LIN {X 0,Y 413.384,Z 401.555,A -85,B 0,C 180,E1 -10493.04,E2 -10493.04} C_VEL
LIN {X 0,Y 413.39,Z 404.987,A -85,B 0,C 180,E1 -10494.691,E2 -10494.691} C_VEL
LIN {X 0,Y 412.815,Z 411.314,A -85,B 0,C 180,E1 -10497.573,E2 -10497.573} C_VEL
LIN {X 0,Y 412.207,Z 419.076,A -85,B 0,C 180,E1 -10500.936,E2 -10500.936} C_VEL
LIN {X 0,Y 411.681,Z 426.853,A -85,B 0,C 180,E1 -10504.197,E2 -10504.197} C_VEL
LIN {X 0,Y 411.179,Z 436.082,A -85,B 0,C 180,E1 -10507.914,E2 -10507.914} C_VEL
LIN {X 0,Y 410.861,Z 444.017,A -85,B 0,C 180,E1 -10511.036,E2 -10511.036} C_VEL
LIN {X 0,Y 410.682,Z 447.705,A -85,B 0,C 180,E1 -10512.405,E2 -10512.405} C_VEL
LIN {X 0,Y 412.802,Z 461.15,A -85,B 0,C 180,E1 -10512.893,E2 -10512.893} C_VEL
LIN {X 0,Y 414.62,Z 474.244,A -85,B 0,C 180,E1 -10513.572,E2 -10513.572} C_VEL
LIN {X 0,Y 414.778,Z 478.671,A -85,B 0,C 180,E1 -10513.831,E2 -10513.831} C_VEL
LIN {X 0,Y 413.979,Z 490.398,A -85,B 0,C 180,E1 -10514.62,E2 -10514.62} C_VEL
LIN {X 0,Y 413.231,Z 501.649,A -85,B 0,C 180,E1 -10515.59,E2 -10515.59} C_VEL
LIN {X 0,Y 412.528,Z 512,A -85,B 0,C 180,E1 -10516.706,E2 -10516.706} C_VEL
LIN {X 0,Y 411.827,Z 521.233,A -85,B 0,C 180,E1 -10517.935,E2 -10517.935} C_VEL
LIN {X 0,Y 411.123,Z 530.239,A -85,B 0,C 180,E1 -10519.413,E2 -10519.413} C_VEL
LIN {X 0,Y 410.679,Z 537.503,A -85,B 0,C 180,E1 -10520.894,E2 -10520.894} C_VEL
LIN {X 0,Y 410.352,Z 542.408,A -85,B 0,C 180,E1 -10522.127,E2 -10522.127} C_VEL
LIN {X 0,Y 410.175,Z 547.189,A -85,B 0,C 180,E1 -10523.608,E2 -10523.608} C_VEL
LIN {X 0,Y 410.096,Z 550.845,A -85,B 0,C 180,E1 -10525.086,E2 -10525.086} C_VEL
LIN {X 0,Y 409.955,Z 552.727,A -85,B 0,C 180,E1 -10526.07,E2 -10526.07} C_VEL
LIN {X 0,Y 410.007,Z 554.15,A -85,B 0,C 180,E1 -10527.054,E2 -10527.054} C_VEL
LIN {X 0,Y 409.988,Z 555.163,A -85,B 0,C 180,E1 -10528.037,E2 -10528.037} C_VEL
LIN {X 0,Y 409.959,Z 555.783,A -85,B 0,C 180,E1 -10529.02,E2 -10529.02} C_VEL
LIN {X 0,Y 409.967,Z 556.008,A -85,B 0,C 180,E1 -10530.002,E2 -10530.002} C_VEL
LIN {X 0,Y 409.959,Z 555.794,A -85,B 0,C 180,E1 -10530.984,E2 -10530.984} C_VEL
LIN {X 0,Y 409.989,Z 555.187,A -85,B 0,C 180,E1 -10531.967,E2 -10531.967} C_VEL
LIN {X 0,Y 410.008,Z 554.186,A -85,B 0,C 180,E1 -10532.949,E2 -10532.949} C_VEL
LIN {X 0,Y 409.955,Z 552.774,A -85,B 0,C 180,E1 -10533.934,E2 -10533.934} C_VEL
LIN {X 0,Y 410.109,Z 549.821,A -85,B 0,C 180,E1 -10535.41,E2 -10535.41} C_VEL
LIN {X 0,Y 410.2,Z 545.812,A -85,B 0,C 180,E1 -10536.89,E2 -10536.89} C_VEL
LIN {X 0,Y 410.553,Z 539.656,A -85,B 0,C 180,E1 -10538.616,E2 -10538.616} C_VEL
LIN {X 0,Y 410.995,Z 532.935,A -85,B 0,C 180,E1 -10540.096,E2 -10540.096} C_VEL
LIN {X 0,Y 411.586,Z 524.602,A -85,B 0,C 180,E1 -10541.576,E2 -10541.576} C_VEL
LIN {X 0,Y 412.261,Z 516.065,A -85,B 0,C 180,E1 -10542.806,E2 -10542.806} C_VEL
LIN {X 0,Y 412.962,Z 505.339,A -85,B 0,C 180,E1 -10544.056,E2 -10544.056} C_VEL
LIN {X 0,Y 413.802,Z 493.67,A -85,B 0,C 180,E1 -10545.139,E2 -10545.139} C_VEL
LIN {X 0,Y 414.646,Z 481.768,A -85,B 0,C 180,E1 -10545.988,E2 -10545.988} C_VEL
LIN {X 0,Y 414.818,Z 475.494,A -85,B 0,C 180,E1 -10546.359,E2 -10546.359} C_VEL
LIN {X 0,Y 413.068,Z 462.585,A -85,B 0,C 180,E1 -10547.042,E2 -10547.042} C_VEL
LIN {X 0,Y 410.836,Z 449.124,A -85,B 0,C 180,E1 -10547.554,E2 -10547.554} C_VEL
LIN {X 0,Y 410.721,Z 447.803,A -85,B 0,C 180,E1 -10547.635,E2 -10547.635} C_VEL
LIN {X 0,Y 411.094,Z 439.097,A -85,B 0,C 180,E1 -10551.041,E2 -10551.041} C_VEL
LIN {X 0,Y 411.483,Z 431.213,A -85,B 0,C 180,E1 -10554.201,E2 -10554.201} C_VEL
LIN {X 0,Y 411.896,Z 424.656,A -85,B 0,C 180,E1 -10556.884,E2 -10556.884} C_VEL
LIN {X 0,Y 412.427,Z 416.854,A -85,B 0,C 180,E1 -10560.18,E2 -10560.18} C_VEL
LIN {X 0,Y 413.084,Z 409.18,A -85,B 0,C 180,E1 -10563.523,E2 -10563.523} C_VEL
LIN {X 0,Y 413.51,Z 403.963,A -85,B 0,C 180,E1 -10565.9,E2 -10565.9} C_VEL
LIN {X 0,Y 413.155,Z 400.089,A -85,B 0,C 180,E1 -10567.763,E2 -10567.763} C_VEL
LIN {X 0,Y 411.926,Z 393.158,A -85,B 0,C 180,E1 -10571.349,E2 -10571.349} C_VEL
LIN {X 0,Y 411.183,Z 389.269,A -85,B 0,C 180,E1 -10573.596,E2 -10573.596} C_VEL
LIN {X 0,Y 411.179,Z 389.27,A -85,B 0,C 180,E1 -10576.867,E2 -10576.867} C_VEL
LIN {X 0,Y 411.215,Z 389.263,A -85,B 0,C 180,E1 -10580.273,E2 -10580.273} C_VEL
LIN {X 0,Y 411.198,Z 389.264,A -85,B 0,C 180,E1 -10583.448,E2 -10583.448} C_VEL
LIN {X 0,Y 411.213,Z 389.265,A -85,B 0,C 180,E1 -10586.874,E2 -10586.874} C_VEL
LIN {X 0,Y 411.239,Z 389.262,A -85,B 0,C 180,E1 -10590.645,E2 -10590.645} C_VEL
LIN {X 0,Y 411.244,Z 389.257,A -85,B 0,C 180,E1 -10593.619,E2 -10593.619} C_VEL
LIN {X 0,Y 411.209,Z 389.265,A -85,B 0,C 180,E1 -10596.853,E2 -10596.853} C_VEL
LIN {X 0,Y 411.221,Z 389.263,A -85,B 0,C 180,E1 -10600.051,E2 -10600.051} C_VEL
LIN {X 0,Y 411.269,Z 389.255,A -85,B 0,C 180,E1 -10603.131,E2 -10603.131} C_VEL
LIN {X 0,Y 411.311,Z 389.25,A -85,B 0,C 180,E1 -10606.896,E2 -10606.896} C_VEL
LIN {X 0,Y 411.298,Z 389.255,A -85,B 0,C 180,E1 -10610.161,E2 -10610.161} C_VEL
LIN {X 0,Y 411.458,Z 389.23,A -85,B 0,C 180,E1 -10613.133,E2 -10613.133} C_VEL
LIN {X 0,Y 411.313,Z 389.249,A -85,B 0,C 180,E1 -10615.099,E2 -10615.099} C_VEL
LIN {X 0,Y 411.516,Z 389.228,A -85,B 0,C 180,E1 -10618.042,E2 -10618.042} C_VEL
LIN {X 0,Y 411.645,Z 389.212,A -85,B 0,C 180,E1 -10620,E2 -10620} C_VEL
LIN {X 0,Y 411.462,Z 389.23,A -85,B 0,C 180,E1 -10622.937,E2 -10622.937} C_VEL
LIN {X 0,Y 411.464,Z 389.23,A -85,B 0,C 180,E1 -10626.867,E2 -10626.867} C_VEL
LIN {X 0,Y 411.36,Z 389.242,A -85,B 0,C 180,E1 -10628.845,E2 -10628.845} C_VEL
LIN {X 0,Y 411.289,Z 389.256,A -85,B 0,C 180,E1 -10631.833,E2 -10631.833} C_VEL
LIN {X 0,Y 411.265,Z 389.255,A -85,B 0,C 180,E1 -10634.852,E2 -10634.852} C_VEL
LIN {X 0,Y 411.258,Z 389.259,A -85,B 0,C 180,E1 -10637.915,E2 -10637.915} C_VEL
LIN {X 0,Y 411.202,Z 389.264,A -85,B 0,C 180,E1 -10641.034,E2 -10641.034} C_VEL
LIN {X 0,Y 411.232,Z 389.26,A -85,B 0,C 180,E1 -10644.215,E2 -10644.215} C_VEL
LIN {X 0,Y 411.265,Z 389.259,A -85,B 0,C 180,E1 -10647.477,E2 -10647.477} C_VEL
LIN {X 0,Y 411.195,Z 389.264,A -85,B 0,C 180,E1 -10650.847,E2 -10650.847} C_VEL
LIN {X 0,Y 411.211,Z 389.262,A -85,B 0,C 180,E1 -10654.333,E2 -10654.333} C_VEL
LIN {X 0,Y 411.2,Z 389.264,A -85,B 0,C 180,E1 -10657.973,E2 -10657.973} C_VEL
LIN {X 0,Y 411.187,Z 389.265,A -85,B 0,C 180,E1 -10660.504,E2 -10660.504} C_VEL
LIN {X 0,Y 411.179,Z 389.269,A -85,B 0,C 180,E1 -10663.133,E2 -10663.133} C_VEL
LIN {X 0,Y 411.173,Z 389.266,A -85,B 0,C 180,E1 -10665.88,E2 -10665.88} C_VEL
LIN {X 0,Y 411.169,Z 389.269,A -85,B 0,C 180,E1 -10668.771,E2 -10668.771} C_VEL
LIN {X 0,Y 411.211,Z 389.262,A -85,B 0,C 180,E1 -10671.83,E2 -10671.83} C_VEL
LIN {X 0,Y 411.216,Z 389.265,A -85,B 0,C 180,E1 -10675.121,E2 -10675.121} C_VEL
LIN {X 0,Y 411.171,Z 389.266,A -85,B 0,C 180,E1 -10678.002,E2 -10678.002} C_VEL
LIN {X 0,Y 411.223,Z 389.261,A -85,B 0,C 180,E1 -10681.409,E2 -10681.409} C_VEL
LIN {X 0,Y 411.243,Z 389.257,A -85,B 0,C 180,E1 -10683.618,E2 -10683.618} C_VEL
LIN {X 0,Y 411.208,Z 389.266,A -85,B 0,C 180,E1 -10686.851,E2 -10686.851} C_VEL
LIN {X 0,Y 411.22,Z 389.261,A -85,B 0,C 180,E1 -10690.049,E2 -10690.049} C_VEL
LIN {X 0,Y 411.268,Z 389.257,A -85,B 0,C 180,E1 -10693.13,E2 -10693.13} C_VEL
LIN {X 0,Y 411.236,Z 389.261,A -85,B 0,C 180,E1 -10696.156,E2 -10696.156} C_VEL
LIN {X 0,Y 411.194,Z 389.266,A -85,B 0,C 180,E1 -10698.163,E2 -10698.163} C_VEL
LIN {X 0,Y 410.866,Z 389.309,A -85,B 0,C 180,E1 -10701.142,E2 -10701.142} C_VEL
LIN {X 0,Y 410.774,Z 389.525,A -85,B 0,C 180,E1 -10702.131,E2 -10702.131} C_VEL
LIN {X 0,Y 410.784,Z 392.396,A -85,B 0,C 180,E1 -10705.091,E2 -10705.091} C_VEL
LIN {X 0,Y 410.551,Z 394.344,A -85,B 0,C 180,E1 -10707.054,E2 -10707.054} C_VEL
LIN {X 0,Y 410.411,Z 397.302,A -85,B 0,C 180,E1 -10709.998,E2 -10709.998} C_VEL
LIN {X 0,Y 410.505,Z 401.242,A -85,B 0,C 180,E1 -10713.925,E2 -10713.925} C_VEL
LIN {X 0,Y 410.425,Z 402.961,A -85,B 0,C 180,E1 -10715.556,E2 -10715.556} C_VEL
LIN {X 0,Y 414.064,Z 417.484,A -85,B 0,C 180,E1 -10716.24,E2 -10716.24} C_VEL
LIN {X 0,Y 415.548,Z 425.03,A -85,B 0,C 180,E1 -10716.675,E2 -10716.675} C_VEL
LIN {X 0,Y 414.873,Z 437.253,A -85,B 0,C 180,E1 -10717.42,E2 -10717.42} C_VEL
LIN {X 0,Y 414.236,Z 448.24,A -85,B 0,C 180,E1 -10718.29,E2 -10718.29} C_VEL
LIN {X 0,Y 413.445,Z 458.989,A -85,B 0,C 180,E1 -10719.36,E2 -10719.36} C_VEL
LIN {X 0,Y 412.757,Z 468.534,A -85,B 0,C 180,E1 -10720.545,E2 -10720.545} C_VEL
LIN {X 0,Y 412.152,Z 476.118,A -85,B 0,C 180,E1 -10721.683,E2 -10721.683} C_VEL
LIN {X 0,Y 411.15,Z 479.89,A -85,B 0,C 180,E1 -10722.305,E2 -10722.305} C_VEL
LIN {X 0,Y 407.883,Z 485.677,A -85,B 0,C 180,E1 -10723.336,E2 -10723.336} C_VEL
LIN {X 0,Y 404.703,Z 490.822,A -85,B 0,C 180,E1 -10724.443,E2 -10724.443} C_VEL
LIN {X 0,Y 403.848,Z 493.53,A -85,B 0,C 180,E1 -10725.177,E2 -10725.177} C_VEL
LIN {X 0,Y 403.486,Z 498.112,A -85,B 0,C 180,E1 -10726.664,E2 -10726.664} C_VEL
LIN {X 0,Y 403.2,Z 501.878,A -85,B 0,C 180,E1 -10728.283,E2 -10728.283} C_VEL
LIN {X 0,Y 403.025,Z 504.16,A -85,B 0,C 180,E1 -10729.668,E2 -10729.668} C_VEL
LIN {X 0,Y 402.881,Z 506,A -85,B 0,C 180,E1 -10731.487,E2 -10731.487} C_VEL
LIN {X 0,Y 402.85,Z 506.437,A -85,B 0,C 180,E1 -10732.567,E2 -10732.567} C_VEL
LIN {X 0,Y 402.857,Z 506.444,A -85,B 0,C 180,E1 -10733.653,E2 -10733.653} C_VEL
LIN {X 0,Y 402.893,Z 505.879,A -85,B 0,C 180,E1 -10734.895,E2 -10734.895} C_VEL
LIN {X 0,Y 402.978,Z 505.025,A -85,B 0,C 180,E1 -10735.846,E2 -10735.846} C_VEL
LIN {X 0,Y 403.169,Z 503.115,A -85,B 0,C 180,E1 -10737.249,E2 -10737.249} C_VEL
LIN {X 0,Y 403.388,Z 500.443,A -85,B 0,C 180,E1 -10738.625,E2 -10738.625} C_VEL
LIN {X 0,Y 403.718,Z 495.928,A -85,B 0,C 180,E1 -10740.318,E2 -10740.318} C_VEL
LIN {X 0,Y 404.191,Z 490.125,A -85,B 0,C 180,E1 -10741.966,E2 -10741.966} C_VEL
LIN {X 0,Y 404.843,Z 482.961,A -85,B 0,C 180,E1 -10743.564,E2 -10743.564} C_VEL
LIN {X 0,Y 405.459,Z 475.593,A -85,B 0,C 180,E1 -10744.887,E2 -10744.887} C_VEL
LIN {X 0,Y 406.229,Z 466.736,A -85,B 0,C 180,E1 -10746.181,E2 -10746.181} C_VEL
LIN {X 0,Y 407.033,Z 456.303,A -85,B 0,C 180,E1 -10747.415,E2 -10747.415} C_VEL
LIN {X 0,Y 407.848,Z 444.851,A -85,B 0,C 180,E1 -10748.492,E2 -10748.492} C_VEL
LIN {X 0,Y 408.543,Z 433.308,A -85,B 0,C 180,E1 -10749.333,E2 -10749.333} C_VEL
LIN {X 0,Y 408.71,Z 425.291,A -85,B 0,C 180,E1 -10749.813,E2 -10749.813} C_VEL
LIN {X 0,Y 405.684,Z 412.827,A -85,B 0,C 180,E1 -10750.529,E2 -10750.529} C_VEL
LIN {X 0,Y 403.305,Z 404.188,A -85,B 0,C 180,E1 -10750.941,E2 -10750.941} C_VEL
LIN {X 0,Y 403.412,Z 400.785,A -85,B 0,C 180,E1 -10754.416,E2 -10754.416} C_VEL
LIN {X 0,Y 403.442,Z 398.12,A -85,B 0,C 180,E1 -10757.204,E2 -10757.204} C_VEL
LIN {X 0,Y 403.54,Z 395.443,A -85,B 0,C 180,E1 -10760.018,E2 -10760.018} C_VEL
LIN {X 0,Y 403.676,Z 391.997,A -85,B 0,C 180,E1 -10763.705,E2 -10763.705} C_VEL
LIN {X 0,Y 403.734,Z 390.847,A -85,B 0,C 180,E1 -10764.939,E2 -10764.939} C_VEL
LIN {X 0,Y 403.891,Z 390.181,A -85,B 0,C 180,E1 -10766.635,E2 -10766.635} C_VEL
LIN {X 0,Y 404.121,Z 390.15,A -85,B 0,C 180,E1 -10769.713,E2 -10769.713} C_VEL
LIN {X 0,Y 404.178,Z 390.14,A -85,B 0,C 180,E1 -10773.122,E2 -10773.122} C_VEL
LIN {X 0,Y 404.167,Z 390.144,A -85,B 0,C 180,E1 -10776.425,E2 -10776.425} C_VEL
LIN {X 0,Y 404.208,Z 390.134,A -85,B 0,C 180,E1 -10779.859,E2 -10779.859} C_VEL
LIN {X 0,Y 404.196,Z 390.139,A -85,B 0,C 180,E1 -10782.992,E2 -10782.992} C_VEL
LIN {X 0,Y 404.262,Z 390.128,A -85,B 0,C 180,E1 -10786.938,E2 -10786.938} C_VEL
LIN {X 0,Y 404.252,Z 390.129,A -85,B 0,C 180,E1 -10789.988,E2 -10789.988} C_VEL
LIN {X 0,Y 404.393,Z 390.11,A -85,B 0,C 180,E1 -10793.013,E2 -10793.013} C_VEL
LIN {X 0,Y 404.272,Z 390.129,A -85,B 0,C 180,E1 -10795.014,E2 -10795.014} C_VEL
LIN {X 0,Y 404.464,Z 390.106,A -85,B 0,C 180,E1 -10798.009,E2 -10798.009} C_VEL
LIN {X 0,Y 404.592,Z 390.088,A -85,B 0,C 180,E1 -10800,E2 -10800} C_VEL
LIN {X 0,Y 404.411,Z 390.11,A -85,B 0,C 180,E1 -10802.989,E2 -10802.989} C_VEL
LIN {X 0,Y 404.391,Z 390.113,A -85,B 0,C 180,E1 -10806.988,E2 -10806.988} C_VEL
LIN {X 0,Y 404.251,Z 390.132,A -85,B 0,C 180,E1 -10810.012,E2 -10810.012} C_VEL
LIN {X 0,Y 404.247,Z 390.132,A -85,B 0,C 180,E1 -10813.212,E2 -10813.212} C_VEL
LIN {X 0,Y 404.196,Z 390.139,A -85,B 0,C 180,E1 -10817.008,E2 -10817.008} C_VEL
LIN {X 0,Y 404.189,Z 390.139,A -85,B 0,C 180,E1 -10820.35,E2 -10820.35} C_VEL
LIN {X 0,Y 404.167,Z 390.144,A -85,B 0,C 180,E1 -10823.575,E2 -10823.575} C_VEL
LIN {X 0,Y 404.179,Z 390.143,A -85,B 0,C 180,E1 -10826.878,E2 -10826.878} C_VEL
LIN {X 0,Y 404.129,Z 390.149,A -85,B 0,C 180,E1 -10830.287,E2 -10830.287} C_VEL
LIN {X 0,Y 404.129,Z 390.147,A -85,B 0,C 180,E1 -10833.814,E2 -10833.814} C_VEL
LIN {X 0,Y 404.126,Z 390.147,A -85,B 0,C 180,E1 -10836.878,E2 -10836.878} C_VEL
LIN {X 0,Y 404.154,Z 390.147,A -85,B 0,C 180,E1 -10840.085,E2 -10840.085} C_VEL
LIN {X 0,Y 404.192,Z 390.146,A -85,B 0,C 180,E1 -10843.094,E2 -10843.094} C_VEL
LIN {X 0,Y 404.219,Z 390.214,A -85,B 0,C 180,E1 -10845.98,E2 -10845.98} C_VEL
LIN {X 0,Y 405.367,Z 396.616,A -85,B 0,C 180,E1 -10849.716,E2 -10849.716} C_VEL
LIN {X 0,Y 406.32,Z 402.279,A -85,B 0,C 180,E1 -10852.747,E2 -10852.747} C_VEL
LIN {X 0,Y 406.437,Z 405.532,A -85,B 0,C 180,E1 -10854.362,E2 -10854.362} C_VEL
LIN {X 0,Y 405.804,Z 412.364,A -85,B 0,C 180,E1 -10857.531,E2 -10857.531} C_VEL
LIN {X 0,Y 405.153,Z 420.058,A -85,B 0,C 180,E1 -10860.944,E2 -10860.944} C_VEL
LIN {X 0,Y 404.633,Z 427.83,A -85,B 0,C 180,E1 -10864.267,E2 -10864.267} C_VEL
LIN {X 0,Y 404.089,Z 437.021,A -85,B 0,C 180,E1 -10868.044,E2 -10868.044} C_VEL
LIN {X 0,Y 403.742,Z 444.938,A -85,B 0,C 180,E1 -10871.217,E2 -10871.217} C_VEL
LIN {X 0,Y 403.641,Z 447.176,A -85,B 0,C 180,E1 -10872.08,E2 -10872.08} C_VEL
LIN {X 0,Y 405.791,Z 460.799,A -85,B 0,C 180,E1 -10872.589,E2 -10872.589} C_VEL
LIN {X 0,Y 407.58,Z 473.449,A -85,B 0,C 180,E1 -10873.259,E2 -10873.259} C_VEL
LIN {X 0,Y 407.981,Z 477.702,A -85,B 0,C 180,E1 -10873.519,E2 -10873.519} C_VEL
LIN {X 0,Y 407.115,Z 489.968,A -85,B 0,C 180,E1 -10874.354,E2 -10874.354} C_VEL
LIN {X 0,Y 406.286,Z 501.704,A -85,B 0,C 180,E1 -10875.386,E2 -10875.386} C_VEL
LIN {X 0,Y 405.587,Z 511.564,A -85,B 0,C 180,E1 -10876.474,E2 -10876.474} C_VEL
LIN {X 0,Y 404.868,Z 520.796,A -85,B 0,C 180,E1 -10877.725,E2 -10877.725} C_VEL
LIN {X 0,Y 404.1,Z 529.801,A -85,B 0,C 180,E1 -10879.227,E2 -10879.227} C_VEL
LIN {X 0,Y 403.61,Z 537.065,A -85,B 0,C 180,E1 -10880.733,E2 -10880.733} C_VEL
LIN {X 0,Y 403.299,Z 541.973,A -85,B 0,C 180,E1 -10881.988,E2 -10881.988} C_VEL
LIN {X 0,Y 403.069,Z 547.202,A -85,B 0,C 180,E1 -10883.652,E2 -10883.652} C_VEL
LIN {X 0,Y 403.008,Z 550.411,A -85,B 0,C 180,E1 -10885,E2 -10885} C_VEL
LIN {X 0,Y 402.877,Z 552.295,A -85,B 0,C 180,E1 -10886.001,E2 -10886.001} C_VEL
LIN {X 0,Y 402.909,Z 553.717,A -85,B 0,C 180,E1 -10887.002,E2 -10887.002} C_VEL
LIN {X 0,Y 402.921,Z 554.733,A -85,B 0,C 180,E1 -10888.003,E2 -10888.003} C_VEL
LIN {X 0,Y 402.884,Z 555.353,A -85,B 0,C 180,E1 -10889.002,E2 -10889.002} C_VEL
LIN {X 0,Y 402.89,Z 555.578,A -85,B 0,C 180,E1 -10890.002,E2 -10890.002} C_VEL
LIN {X 0,Y 402.921,Z 554.757,A -85,B 0,C 180,E1 -10892.001,E2 -10892.001} C_VEL
LIN {X 0,Y 402.91,Z 553.754,A -85,B 0,C 180,E1 -10893.001,E2 -10893.001} C_VEL
LIN {X 0,Y 402.878,Z 552.343,A -85,B 0,C 180,E1 -10894.003,E2 -10894.003} C_VEL
LIN {X 0,Y 403.007,Z 549.387,A -85,B 0,C 180,E1 -10895.506,E2 -10895.506} C_VEL
LIN {X 0,Y 403.118,Z 545.377,A -85,B 0,C 180,E1 -10897.012,E2 -10897.012} C_VEL
LIN {X 0,Y 403.518,Z 539.219,A -85,B 0,C 180,E1 -10898.768,E2 -10898.768} C_VEL
LIN {X 0,Y 403.967,Z 532.495,A -85,B 0,C 180,E1 -10900.274,E2 -10900.274} C_VEL
LIN {X 0,Y 404.6,Z 524.161,A -85,B 0,C 180,E1 -10901.779,E2 -10901.779} C_VEL
LIN {X 0,Y 405.266,Z 515.617,A -85,B 0,C 180,E1 -10903.031,E2 -10903.031} C_VEL
LIN {X 0,Y 405.984,Z 505.786,A -85,B 0,C 180,E1 -10904.205,E2 -10904.205} C_VEL
LIN {X 0,Y 406.807,Z 494.65,A -85,B 0,C 180,E1 -10905.277,E2 -10905.277} C_VEL
LIN {X 0,Y 407.657,Z 483.352,A -85,B 0,C 180,E1 -10906.134,E2 -10906.134} C_VEL
LIN {X 0,Y 407.882,Z 475.699,A -85,B 0,C 180,E1 -10906.607,E2 -10906.607} C_VEL
LIN {X 0,Y 406.106,Z 462.732,A -85,B 0,C 180,E1 -10907.316,E2 -10907.316} C_VEL
LIN {X 0,Y 403.985,Z 449.659,A -85,B 0,C 180,E1 -10907.838,E2 -10907.838} C_VEL
LIN {X 0,Y 403.644,Z 447.403,A -85,B 0,C 180,E1 -10907.938,E2 -10907.938} C_VEL
LIN {X 0,Y 404.013,Z 440.038,A -85,B 0,C 180,E1 -10910.894,E2 -10910.894} C_VEL
LIN {X 0,Y 404.394,Z 432.159,A -85,B 0,C 180,E1 -10914.106,E2 -10914.106} C_VEL
LIN {X 0,Y 404.897,Z 424.569,A -85,B 0,C 180,E1 -10917.284,E2 -10917.284} C_VEL
LIN {X 0,Y 405.5,Z 416.561,A -85,B 0,C 180,E1 -10920.751,E2 -10920.751} C_VEL
LIN {X 0,Y 406.127,Z 409.667,A -85,B 0,C 180,E1 -10923.835,E2 -10923.835} C_VEL
LIN {X 0,Y 406.507,Z 404.99,A -85,B 0,C 180,E1 -10926.004,E2 -10926.004} C_VEL
LIN {X 0,Y 406.143,Z 401.148,A -85,B 0,C 180,E1 -10927.902,E2 -10927.902} C_VEL
LIN {X 0,Y 405.017,Z 394.766,A -85,B 0,C 180,E1 -10931.255,E2 -10931.255} C_VEL
LIN {X 0,Y 404.143,Z 390.145,A -85,B 0,C 180,E1 -10933.875,E2 -10933.875} C_VEL
LIN {X 0,Y 404.142,Z 390.146,A -85,B 0,C 180,E1 -10937.296,E2 -10937.296} C_VEL
LIN {X 0,Y 404.176,Z 390.14,A -85,B 0,C 180,E1 -10939.956,E2 -10939.956} C_VEL
LIN {X 0,Y 404.142,Z 390.145,A -85,B 0,C 180,E1 -10943.126,E2 -10943.126} C_VEL
LIN {X 0,Y 404.15,Z 390.142,A -85,B 0,C 180,E1 -10946.188,E2 -10946.188} C_VEL
LIN {X 0,Y 404.152,Z 390.14,A -85,B 0,C 180,E1 -10949.715,E2 -10949.715} C_VEL
LIN {X 0,Y 404.202,Z 390.136,A -85,B 0,C 180,E1 -10953.123,E2 -10953.123} C_VEL
LIN {X 0,Y 404.183,Z 390.137,A -85,B 0,C 180,E1 -10955.335,E2 -10955.335} C_VEL
LIN {X 0,Y 404.145,Z 390.146,A -85,B 0,C 180,E1 -10958.581,E2 -10958.581} C_VEL
LIN {X 0,Y 404.216,Z 390.133,A -85,B 0,C 180,E1 -10961.762,E2 -10961.762} C_VEL
LIN {X 0,Y 404.212,Z 390.135,A -85,B 0,C 180,E1 -10964.882,E2 -10964.882} C_VEL
LIN {X 0,Y 404.262,Z 390.13,A -85,B 0,C 180,E1 -10967.959,E2 -10967.959} C_VEL
LIN {X 0,Y 404.411,Z 390.113,A -85,B 0,C 180,E1 -10972.129,E2 -10972.129} C_VEL
LIN {X 0,Y 404.425,Z 390.111,A -85,B 0,C 180,E1 -10974.015,E2 -10974.015} C_VEL
LIN {X 0,Y 404.485,Z 390.103,A -85,B 0,C 180,E1 -10978.008,E2 -10978.008} C_VEL
LIN {X 0,Y 404.614,Z 390.087,A -85,B 0,C 180,E1 -10980,E2 -10980} C_VEL
LIN {X 0,Y 404.42,Z 390.107,A -85,B 0,C 180,E1 -10982.988,E2 -10982.988} C_VEL
LIN {X 0,Y 404.415,Z 390.107,A -85,B 0,C 180,E1 -10986.987,E2 -10986.987} C_VEL
LIN {X 0,Y 404.264,Z 390.131,A -85,B 0,C 180,E1 -10990.012,E2 -10990.012} C_VEL
LIN {X 0,Y 404.272,Z 390.126,A -85,B 0,C 180,E1 -10993.211,E2 -10993.211} C_VEL
LIN {X 0,Y 404.222,Z 390.132,A -85,B 0,C 180,E1 -10997.007,E2 -10997.007} C_VEL
LIN {X 0,Y 404.169,Z 390.139,A -85,B 0,C 180,E1 -11000.351,E2 -11000.351} C_VEL
LIN {X 0,Y 404.175,Z 390.142,A -85,B 0,C 180,E1 -11003.574,E2 -11003.574} C_VEL
LIN {X 0,Y 404.19,Z 390.14,A -85,B 0,C 180,E1 -11005.766,E2 -11005.766} C_VEL
LIN {X 0,Y 404.201,Z 390.136,A -85,B 0,C 180,E1 -11007.999,E2 -11007.999} C_VEL
LIN {X 0,Y 404.145,Z 390.146,A -85,B 0,C 180,E1 -11011.557,E2 -11011.557} C_VEL
LIN {X 0,Y 404.19,Z 390.139,A -85,B 0,C 180,E1 -11015.016,E2 -11015.016} C_VEL
LIN {X 0,Y 404.16,Z 390.141,A -85,B 0,C 180,E1 -11018.756,E2 -11018.756} C_VEL
LIN {X 0,Y 404.129,Z 390.146,A -85,B 0,C 180,E1 -11021.599,E2 -11021.599} C_VEL
LIN {X 0,Y 404.151,Z 390.141,A -85,B 0,C 180,E1 -11024.521,E2 -11024.521} C_VEL
LIN {X 0,Y 404.142,Z 390.146,A -85,B 0,C 180,E1 -11027.295,E2 -11027.295} C_VEL
LIN {X 0,Y 404.175,Z 390.138,A -85,B 0,C 180,E1 -11029.955,E2 -11029.955} C_VEL
LIN {X 0,Y 404.142,Z 390.146,A -85,B 0,C 180,E1 -11033.124,E2 -11033.124} C_VEL
LIN {X 0,Y 404.15,Z 390.141,A -85,B 0,C 180,E1 -11036.187,E2 -11036.187} C_VEL
LIN {X 0,Y 404.151,Z 390.141,A -85,B 0,C 180,E1 -11039.714,E2 -11039.714} C_VEL
LIN {X 0,Y 404.201,Z 390.138,A -85,B 0,C 180,E1 -11043.122,E2 -11043.122} C_VEL
LIN {X 0,Y 404.182,Z 390.138,A -85,B 0,C 180,E1 -11045.333,E2 -11045.333} C_VEL
LIN {X 0,Y 404.144,Z 390.146,A -85,B 0,C 180,E1 -11048.579,E2 -11048.579} C_VEL
LIN {X 0,Y 404.215,Z 390.133,A -85,B 0,C 180,E1 -11051.761,E2 -11051.761} C_VEL
LIN {X 0,Y 404.21,Z 390.137,A -85,B 0,C 180,E1 -11054.881,E2 -11054.881} C_VEL
LIN {X 0,Y 404.165,Z 390.14,A -85,B 0,C 180,E1 -11057.954,E2 -11057.954} C_VEL
LIN {X 0,Y 403.858,Z 390.182,A -85,B 0,C 180,E1 -11060.988,E2 -11060.988} C_VEL
LIN {X 0,Y 403.721,Z 390.231,A -85,B 0,C 180,E1 -11061.993,E2 -11061.993} C_VEL
LIN {X 0,Y 403.735,Z 393.111,A -85,B 0,C 180,E1 -11065.005,E2 -11065.005} C_VEL
LIN {X 0,Y 403.509,Z 395.091,A -85,B 0,C 180,E1 -11067.003,E2 -11067.003} C_VEL
LIN {X 0,Y 403.352,Z 398.094,A -85,B 0,C 180,E1 -11069.998,E2 -11069.998} C_VEL
LIN {X 0,Y 403.435,Z 401.056,A -85,B 0,C 180,E1 -11072.994,E2 -11072.994} C_VEL
LIN {X 0,Y 403.359,Z 403.34,A -85,B 0,C 180,E1 -11075.246,E2 -11075.246} C_VEL
LIN {X 0,Y 406.893,Z 417.253,A -85,B 0,C 180,E1 -11075.915,E2 -11075.915} C_VEL
LIN {X 0,Y 408.648,Z 425.75,A -85,B 0,C 180,E1 -11076.416,E2 -11076.416} C_VEL
LIN {X 0,Y 408.042,Z 437.83,A -85,B 0,C 180,E1 -11077.171,E2 -11077.171} C_VEL
LIN {X 0,Y 407.365,Z 448.794,A -85,B 0,C 180,E1 -11078.056,E2 -11078.056} C_VEL
LIN {X 0,Y 406.593,Z 459.049,A -85,B 0,C 180,E1 -11079.09,E2 -11079.09} C_VEL
LIN {X 0,Y 405.901,Z 468.13,A -85,B 0,C 180,E1 -11080.221,E2 -11080.221} C_VEL
LIN {X 0,Y 405.178,Z 476.751,A -85,B 0,C 180,E1 -11081.529,E2 -11081.529} C_VEL
LIN {X 0,Y 404.509,Z 484.878,A -85,B 0,C 180,E1 -11083.051,E2 -11083.051} C_VEL
LIN {X 0,Y 403.993,Z 491.499,A -85,B 0,C 180,E1 -11084.608,E2 -11084.608} C_VEL
LIN {X 0,Y 403.848,Z 493.53,A -85,B 0,C 180,E1 -11085.177,E2 -11085.177} C_VEL
LIN {X 0,Y 402.993,Z 496.078,A -85,B 0,C 180,E1 -11085.931,E2 -11085.931} C_VEL
LIN {X 0,Y 399.834,Z 499.728,A -85,B 0,C 180,E1 -11087.169,E2 -11087.169} C_VEL
LIN {X 0,Y 396.728,Z 502.721,A -85,B 0,C 180,E1 -11088.458,E2 -11088.458} C_VEL
LIN {X 0,Y 395.963,Z 504.065,A -85,B 0,C 180,E1 -11089.281,E2 -11089.281} C_VEL
LIN {X 0,Y 395.82,Z 505.911,A -85,B 0,C 180,E1 -11090.798,E2 -11090.798} C_VEL
LIN {X 0,Y 395.787,Z 506.87,A -85,B 0,C 180,E1 -11092.577,E2 -11092.577} C_VEL
LIN {X 0,Y 395.776,Z 506.754,A -85,B 0,C 180,E1 -11094.103,E2 -11094.103} C_VEL
LIN {X 0,Y 395.855,Z 506.098,A -85,B 0,C 180,E1 -11095.217,E2 -11095.217} C_VEL
LIN {X 0,Y 395.956,Z 504.986,A -85,B 0,C 180,E1 -11096.34,E2 -11096.34} C_VEL
LIN {X 0,Y 396.239,Z 502.315,A -85,B 0,C 180,E1 -11098.032,E2 -11098.032} C_VEL
LIN {X 0,Y 396.53,Z 498.365,A -85,B 0,C 180,E1 -11099.75,E2 -11099.75} C_VEL
LIN {X 0,Y 396.96,Z 493.376,A -85,B 0,C 180,E1 -11101.37,E2 -11101.37} C_VEL
LIN {X 0,Y 397.552,Z 487.256,A -85,B 0,C 180,E1 -11102.926,E2 -11102.926} C_VEL
LIN {X 0,Y 398.151,Z 480.117,A -85,B 0,C 180,E1 -11104.389,E2 -11104.389} C_VEL
LIN {X 0,Y 398.993,Z 471.02,A -85,B 0,C 180,E1 -11105.879,E2 -11105.879} C_VEL
LIN {X 0,Y 399.821,Z 461.214,A -85,B 0,C 180,E1 -11107.171,E2 -11107.171} C_VEL
LIN {X 0,Y 400.62,Z 451.62,A -85,B 0,C 180,E1 -11108.195,E2 -11108.195} C_VEL
LIN {X 0,Y 401.439,Z 440.118,A -85,B 0,C 180,E1 -11109.178,E2 -11109.178} C_VEL
LIN {X 0,Y 402.044,Z 427.299,A -85,B 0,C 180,E1 -11110.016,E2 -11110.016} C_VEL
LIN {X 0,Y 399.094,Z 414.764,A -85,B 0,C 180,E1 -11110.78,E2 -11110.78} C_VEL
LIN {X 0,Y 396.262,Z 404.634,A -85,B 0,C 180,E1 -11111.281,E2 -11111.281} C_VEL
LIN {X 0,Y 396.361,Z 401.217,A -85,B 0,C 180,E1 -11114.826,E2 -11114.826} C_VEL
LIN {X 0,Y 396.417,Z 398.088,A -85,B 0,C 180,E1 -11118.121,E2 -11118.121} C_VEL
LIN {X 0,Y 396.52,Z 394.824,A -85,B 0,C 180,E1 -11121.659,E2 -11121.659} C_VEL
LIN {X 0,Y 396.667,Z 392.103,A -85,B 0,C 180,E1 -11124.583,E2 -11124.583} C_VEL
LIN {X 0,Y 396.68,Z 391.311,A -85,B 0,C 180,E1 -11125.463,E2 -11125.463} C_VEL
LIN {X 0,Y 397.013,Z 391.038,A -85,B 0,C 180,E1 -11128.174,E2 -11128.174} C_VEL
LIN {X 0,Y 397.098,Z 391.022,A -85,B 0,C 180,E1 -11131.455,E2 -11131.455} C_VEL
LIN {X 0,Y 397.135,Z 391.018,A -85,B 0,C 180,E1 -11134.486,E2 -11134.486} C_VEL
LIN {X 0,Y 397.158,Z 391.015,A -85,B 0,C 180,E1 -11138.185,E2 -11138.185} C_VEL
LIN {X 0,Y 397.152,Z 391.015,A -85,B 0,C 180,E1 -11141.426,E2 -11141.426} C_VEL
LIN {X 0,Y 397.16,Z 391.014,A -85,B 0,C 180,E1 -11144.607,E2 -11144.607} C_VEL
LIN {X 0,Y 397.21,Z 391.007,A -85,B 0,C 180,E1 -11147.742,E2 -11147.742} C_VEL
LIN {X 0,Y 397.375,Z 390.986,A -85,B 0,C 180,E1 -11152.04,E2 -11152.04} C_VEL
LIN {X 0,Y 397.244,Z 391.004,A -85,B 0,C 180,E1 -11154.925,E2 -11154.925} C_VEL
LIN {X 0,Y 397.432,Z 390.982,A -85,B 0,C 180,E1 -11157.973,E2 -11157.973} C_VEL
LIN {X 0,Y 397.562,Z 390.963,A -85,B 0,C 180,E1 -11160,E2 -11160} C_VEL
LIN {X 0,Y 397.369,Z 390.988,A -85,B 0,C 180,E1 -11163.042,E2 -11163.042} C_VEL
LIN {X 0,Y 397.344,Z 390.991,A -85,B 0,C 180,E1 -11167.112,E2 -11167.112} C_VEL
LIN {X 0,Y 397.209,Z 391.01,A -85,B 0,C 180,E1 -11170.191,E2 -11170.191} C_VEL
LIN {X 0,Y 397.207,Z 391.008,A -85,B 0,C 180,E1 -11173.322,E2 -11173.322} C_VEL
LIN {X 0,Y 397.163,Z 391.015,A -85,B 0,C 180,E1 -11177.156,E2 -11177.156} C_VEL
LIN {X 0,Y 397.14,Z 391.018,A -85,B 0,C 180,E1 -11180.728,E2 -11180.728} C_VEL
LIN {X 0,Y 397.124,Z 391.022,A -85,B 0,C 180,E1 -11184.019,E2 -11184.019} C_VEL
LIN {X 0,Y 397.177,Z 391.015,A -85,B 0,C 180,E1 -11187.392,E2 -11187.392} C_VEL
LIN {X 0,Y 397.062,Z 391.029,A -85,B 0,C 180,E1 -11190.884,E2 -11190.884} C_VEL
LIN {X 0,Y 397.11,Z 391.022,A -85,B 0,C 180,E1 -11194.495,E2 -11194.495} C_VEL
LIN {X 0,Y 397.095,Z 391.024,A -85,B 0,C 180,E1 -11198.276,E2 -11198.276} C_VEL
LIN {X 0,Y 397.144,Z 391.022,A -85,B 0,C 180,E1 -11201.995,E2 -11201.995} C_VEL
LIN {X 0,Y 397.17,Z 391.082,A -85,B 0,C 180,E1 -11205.569,E2 -11205.569} C_VEL
LIN {X 0,Y 398.022,Z 396.038,A -85,B 0,C 180,E1 -11208.573,E2 -11208.573} C_VEL
LIN {X 0,Y 399.129,Z 402.093,A -85,B 0,C 180,E1 -11211.958,E2 -11211.958} C_VEL
LIN {X 0,Y 399.47,Z 406.118,A -85,B 0,C 180,E1 -11214.027,E2 -11214.027} C_VEL
LIN {X 0,Y 398.915,Z 412.102,A -85,B 0,C 180,E1 -11216.9,E2 -11216.9} C_VEL
LIN {X 0,Y 398.189,Z 419.758,A -85,B 0,C 180,E1 -11220.386,E2 -11220.386} C_VEL
LIN {X 0,Y 397.657,Z 427.498,A -85,B 0,C 180,E1 -11223.782,E2 -11223.782} C_VEL
LIN {X 0,Y 397.122,Z 435.319,A -85,B 0,C 180,E1 -11227.089,E2 -11227.089} C_VEL
LIN {X 0,Y 396.721,Z 444.514,A -85,B 0,C 180,E1 -11230.871,E2 -11230.871} C_VEL
LIN {X 0,Y 396.597,Z 446.645,A -85,B 0,C 180,E1 -11231.736,E2 -11231.736} C_VEL
LIN {X 0,Y 398.896,Z 460.907,A -85,B 0,C 180,E1 -11232.294,E2 -11232.294} C_VEL
LIN {X 0,Y 400.636,Z 473.751,A -85,B 0,C 180,E1 -11232.998,E2 -11232.998} C_VEL
LIN {X 0,Y 401.026,Z 479.493,A -85,B 0,C 180,E1 -11233.367,E2 -11233.367} C_VEL
LIN {X 0,Y 400.139,Z 491.152,A -85,B 0,C 180,E1 -11234.205,E2 -11234.205} C_VEL
LIN {X 0,Y 399.255,Z 502.632,A -85,B 0,C 180,E1 -11235.267,E2 -11235.267} C_VEL
LIN {X 0,Y 398.455,Z 513.253,A -85,B 0,C 180,E1 -11236.508,E2 -11236.508} C_VEL
LIN {X 0,Y 397.739,Z 522.003,A -85,B 0,C 180,E1 -11237.76,E2 -11237.76} C_VEL
LIN {X 0,Y 396.978,Z 530.698,A -85,B 0,C 180,E1 -11239.289,E2 -11239.289} C_VEL
LIN {X 0,Y 396.496,Z 537.664,A -85,B 0,C 180,E1 -11240.823,E2 -11240.823} C_VEL
LIN {X 0,Y 396.138,Z 543.253,A -85,B 0,C 180,E1 -11242.356,E2 -11242.356} C_VEL
LIN {X 0,Y 395.949,Z 547.646,A -85,B 0,C 180,E1 -11243.889,E2 -11243.889} C_VEL
LIN {X 0,Y 395.921,Z 549.978,A -85,B 0,C 180,E1 -11244.91,E2 -11244.91} C_VEL
LIN {X 0,Y 395.802,Z 551.863,A -85,B 0,C 180,E1 -11245.929,E2 -11245.929} C_VEL
LIN {X 0,Y 395.812,Z 553.284,A -85,B 0,C 180,E1 -11246.949,E2 -11246.949} C_VEL
LIN {X 0,Y 395.854,Z 554.303,A -85,B 0,C 180,E1 -11247.967,E2 -11247.967} C_VEL
LIN {X 0,Y 395.813,Z 554.924,A -85,B 0,C 180,E1 -11248.985,E2 -11248.985} C_VEL
LIN {X 0,Y 395.815,Z 555.148,A -85,B 0,C 180,E1 -11250.002,E2 -11250.002} C_VEL
LIN {X 0,Y 395.855,Z 554.327,A -85,B 0,C 180,E1 -11252.037,E2 -11252.037} C_VEL
LIN {X 0,Y 395.813,Z 553.323,A -85,B 0,C 180,E1 -11253.055,E2 -11253.055} C_VEL
LIN {X 0,Y 395.803,Z 551.912,A -85,B 0,C 180,E1 -11254.075,E2 -11254.075} C_VEL
LIN {X 0,Y 395.908,Z 548.952,A -85,B 0,C 180,E1 -11255.605,E2 -11255.605} C_VEL
LIN {X 0,Y 396.063,Z 544.943,A -85,B 0,C 180,E1 -11257.137,E2 -11257.137} C_VEL
LIN {X 0,Y 396.46,Z 538.781,A -85,B 0,C 180,E1 -11258.925,E2 -11258.925} C_VEL
LIN {X 0,Y 396.915,Z 532.054,A -85,B 0,C 180,E1 -11260.458,E2 -11260.458} C_VEL
LIN {X 0,Y 397.595,Z 523.719,A -85,B 0,C 180,E1 -11261.989,E2 -11261.989} C_VEL
LIN {X 0,Y 398.301,Z 515.171,A -85,B 0,C 180,E1 -11263.263,E2 -11263.263} C_VEL
LIN {X 0,Y 399.097,Z 504.859,A -85,B 0,C 180,E1 -11264.508,E2 -11264.508} C_VEL
LIN {X 0,Y 399.944,Z 494.199,A -85,B 0,C 180,E1 -11265.546,E2 -11265.546} C_VEL
LIN {X 0,Y 400.824,Z 482.989,A -85,B 0,C 180,E1 -11266.41,E2 -11266.41} C_VEL
LIN {X 0,Y 401.098,Z 477.767,A -85,B 0,C 180,E1 -11266.746,E2 -11266.746} C_VEL
LIN {X 0,Y 399.452,Z 464.949,A -85,B 0,C 180,E1 -11267.496,E2 -11267.496} C_VEL
LIN {X 0,Y 397.268,Z 451.221,A -85,B 0,C 180,E1 -11268.089,E2 -11268.089} C_VEL
LIN {X 0,Y 396.609,Z 447.084,A -85,B 0,C 180,E1 -11268.234,E2 -11268.234} C_VEL
LIN {X 0,Y 397.042,Z 438.345,A -85,B 0,C 180,E1 -11271.823,E2 -11271.823} C_VEL
LIN {X 0,Y 397.628,Z 429.242,A -85,B 0,C 180,E1 -11275.655,E2 -11275.655} C_VEL
LIN {X 0,Y 398.174,Z 421.406,A -85,B 0,C 180,E1 -11279.04,E2 -11279.04} C_VEL
LIN {X 0,Y 398.774,Z 414.326,A -85,B 0,C 180,E1 -11282.226,E2 -11282.226} C_VEL
LIN {X 0,Y 399.456,Z 407.289,A -85,B 0,C 180,E1 -11285.494,E2 -11285.494} C_VEL
LIN {X 0,Y 399.466,Z 404.726,A -85,B 0,C 180,E1 -11286.741,E2 -11286.741} C_VEL
LIN {X 0,Y 398.668,Z 399.608,A -85,B 0,C 180,E1 -11289.394,E2 -11289.394} C_VEL
LIN {X 0,Y 397.56,Z 393.337,A -85,B 0,C 180,E1 -11292.851,E2 -11292.851} C_VEL
LIN {X 0,Y 397.106,Z 391.023,A -85,B 0,C 180,E1 -11294.271,E2 -11294.271} C_VEL
LIN {X 0,Y 397.075,Z 391.027,A -85,B 0,C 180,E1 -11297.733,E2 -11297.733} C_VEL
LIN {X 0,Y 397.133,Z 391.018,A -85,B 0,C 180,E1 -11301.14,E2 -11301.14} C_VEL
LIN {X 0,Y 397.125,Z 391.019,A -85,B 0,C 180,E1 -11304.497,E2 -11304.497} C_VEL
LIN {X 0,Y 397.084,Z 391.021,A -85,B 0,C 180,E1 -11307.929,E2 -11307.929} C_VEL
LIN {X 0,Y 397.128,Z 391.015,A -85,B 0,C 180,E1 -11311.457,E2 -11311.457} C_VEL
LIN {X 0,Y 397.159,Z 391.016,A -85,B 0,C 180,E1 -11314.488,E2 -11314.488} C_VEL
LIN {X 0,Y 397.115,Z 391.018,A -85,B 0,C 180,E1 -11317.086,E2 -11317.086} C_VEL
LIN {X 0,Y 397.154,Z 391.016,A -85,B 0,C 180,E1 -11320.353,E2 -11320.353} C_VEL
LIN {X 0,Y 397.173,Z 391.01,A -85,B 0,C 180,E1 -11323.553,E2 -11323.553} C_VEL
LIN {X 0,Y 397.235,Z 391.005,A -85,B 0,C 180,E1 -11326.703,E2 -11326.703} C_VEL
LIN {X 0,Y 397.223,Z 391.005,A -85,B 0,C 180,E1 -11329.809,E2 -11329.809} C_VEL
LIN {X 0,Y 397.355,Z 390.987,A -85,B 0,C 180,E1 -11332.888,E2 -11332.888} C_VEL
LIN {X 0,Y 397.257,Z 391,A -85,B 0,C 180,E1 -11334.925,E2 -11334.925} C_VEL
LIN {X 0,Y 397.454,Z 390.979,A -85,B 0,C 180,E1 -11337.973,E2 -11337.973} C_VEL
LIN {X 0,Y 397.584,Z 390.963,A -85,B 0,C 180,E1 -11340,E2 -11340} C_VEL
LIN {X 0,Y 397.379,Z 390.984,A -85,B 0,C 180,E1 -11343.041,E2 -11343.041} C_VEL
LIN {X 0,Y 397.368,Z 390.985,A -85,B 0,C 180,E1 -11347.112,E2 -11347.112} C_VEL
LIN {X 0,Y 397.223,Z 391.007,A -85,B 0,C 180,E1 -11350.191,E2 -11350.191} C_VEL
LIN {X 0,Y 397.233,Z 391.004,A -85,B 0,C 180,E1 -11353.321,E2 -11353.321} C_VEL
LIN {X 0,Y 397.188,Z 391.009,A -85,B 0,C 180,E1 -11357.155,E2 -11357.155} C_VEL
LIN {X 0,Y 397.108,Z 391.018,A -85,B 0,C 180,E1 -11360.73,E2 -11360.73} C_VEL
LIN {X 0,Y 397.139,Z 391.016,A -85,B 0,C 180,E1 -11364.018,E2 -11364.018} C_VEL
LIN {X 0,Y 397.2,Z 391.011,A -85,B 0,C 180,E1 -11367.39,E2 -11367.39} C_VEL
LIN {X 0,Y 397.084,Z 391.022,A -85,B 0,C 180,E1 -11370.882,E2 -11370.882} C_VEL
LIN {X 0,Y 397.131,Z 391.015,A -85,B 0,C 180,E1 -11374.493,E2 -11374.493} C_VEL
LIN {X 0,Y 397.108,Z 391.018,A -85,B 0,C 180,E1 -11378.274,E2 -11378.274} C_VEL
LIN {X 0,Y 397.094,Z 391.022,A -85,B 0,C 180,E1 -11380.908,E2 -11380.908} C_VEL
LIN {X 0,Y 397.107,Z 391.02,A -85,B 0,C 180,E1 -11383.648,E2 -11383.648} C_VEL
LIN {X 0,Y 397.107,Z 391.018,A -85,B 0,C 180,E1 -11386.52,E2 -11386.52} C_VEL
LIN {X 0,Y 397.12,Z 391.017,A -85,B 0,C 180,E1 -11390.422,E2 -11390.422} C_VEL
LIN {X 0,Y 397.114,Z 391.018,A -85,B 0,C 180,E1 -11394.264,E2 -11394.264} C_VEL
LIN {X 0,Y 397.12,Z 391.02,A -85,B 0,C 180,E1 -11396.726,E2 -11396.726} C_VEL
LIN {X 0,Y 397.13,Z 391.016,A -85,B 0,C 180,E1 -11400.295,E2 -11400.295} C_VEL
LIN {X 0,Y 397.2,Z 391.01,A -85,B 0,C 180,E1 -11402.609,E2 -11402.609} C_VEL
LIN {X 0,Y 397.138,Z 391.014,A -85,B 0,C 180,E1 -11405.98,E2 -11405.98} C_VEL
LIN {X 0,Y 397.144,Z 391.013,A -85,B 0,C 180,E1 -11409.703,E2 -11409.703} C_VEL
LIN {X 0,Y 397.186,Z 391.012,A -85,B 0,C 180,E1 -11412.843,E2 -11412.843} C_VEL
LIN {X 0,Y 397.171,Z 391.01,A -85,B 0,C 180,E1 -11415.655,E2 -11415.655} C_VEL
LIN {X 0,Y 397.127,Z 391.016,A -85,B 0,C 180,E1 -11417.737,E2 -11417.737} C_VEL
LIN {X 0,Y 396.827,Z 391.058,A -85,B 0,C 180,E1 -11420.826,E2 -11420.826} C_VEL
LIN {X 0,Y 396.697,Z 391.076,A -85,B 0,C 180,E1 -11421.85,E2 -11421.85} C_VEL
LIN {X 0,Y 396.688,Z 393.859,A -85,B 0,C 180,E1 -11424.916,E2 -11424.916} C_VEL
LIN {X 0,Y 396.469,Z 395.834,A -85,B 0,C 180,E1 -11426.95,E2 -11426.95} C_VEL
LIN {X 0,Y 396.287,Z 398.835,A -85,B 0,C 180,E1 -11429.998,E2 -11429.998} C_VEL
LIN {X 0,Y 396.39,Z 401.899,A -85,B 0,C 180,E1 -11433.047,E2 -11433.047} C_VEL
LIN {X 0,Y 396.332,Z 403.768,A -85,B 0,C 180,E1 -11434.925,E2 -11434.925} C_VEL
LIN {X 0,Y 400.021,Z 418.073,A -85,B 0,C 180,E1 -11435.638,E2 -11435.638} C_VEL
LIN {X 0,Y 401.872,Z 427.426,A -85,B 0,C 180,E1 -11436.21,E2 -11436.21} C_VEL
LIN {X 0,Y 401.214,Z 438.41,A -85,B 0,C 180,E1 -11436.915,E2 -11436.915} C_VEL
LIN {X 0,Y 400.49,Z 449.357,A -85,B 0,C 180,E1 -11437.814,E2 -11437.814} C_VEL
LIN {X 0,Y 399.723,Z 459.413,A -85,B 0,C 180,E1 -11438.848,E2 -11438.848} C_VEL
LIN {X 0,Y 398.889,Z 469.551,A -85,B 0,C 180,E1 -11440.146,E2 -11440.146} C_VEL
LIN {X 0,Y 398.162,Z 477.857,A -85,B 0,C 180,E1 -11441.451,E2 -11441.451} C_VEL
LIN {X 0,Y 397.473,Z 485.983,A -85,B 0,C 180,E1 -11443.027,E2 -11443.027} C_VEL
LIN {X 0,Y 397.019,Z 491.474,A -85,B 0,C 180,E1 -11444.347,E2 -11444.347} C_VEL
LIN {X 0,Y 396.588,Z 496.814,A -85,B 0,C 180,E1 -11445.94,E2 -11445.94} C_VEL
LIN {X 0,Y 396.275,Z 500.929,A -85,B 0,C 180,E1 -11447.545,E2 -11447.545} C_VEL
LIN {X 0,Y 395.963,Z 504.065,A -85,B 0,C 180,E1 -11449.281,E2 -11449.281} C_VEL
LIN {X 0,Y 395.228,Z 505.273,A -85,B 0,C 180,E1 -11450.113,E2 -11450.113} C_VEL
LIN {X 0,Y 392.276,Z 506.696,A -85,B 0,C 180,E1 -11451.475,E2 -11451.475} C_VEL
LIN {X 0,Y 389.814,Z 507.274,A -85,B 0,C 180,E1 -11452.584,E2 -11452.584} C_VEL
LIN {X 0,Y 388.763,Z 507.339,A -85,B 0,C 180,E1 -11453.444,E2 -11453.444} C_VEL
LIN {X 0,Y 388.68,Z 507.253,A -85,B 0,C 180,E1 -11453.735,E2 -11453.735} C_VEL
LIN {X 0,Y 388.778,Z 506.484,A -85,B 0,C 180,E1 -11455.33,E2 -11455.33} C_VEL
LIN {X 0,Y 388.941,Z 504.819,A -85,B 0,C 180,E1 -11456.852,E2 -11456.852} C_VEL
LIN {X 0,Y 389.256,Z 501.847,A -85,B 0,C 180,E1 -11458.582,E2 -11458.582} C_VEL
LIN {X 0,Y 389.611,Z 497.581,A -85,B 0,C 180,E1 -11460.334,E2 -11460.334} C_VEL
LIN {X 0,Y 390.148,Z 491.586,A -85,B 0,C 180,E1 -11462.151,E2 -11462.151} C_VEL
LIN {X 0,Y 390.88,Z 484.249,A -85,B 0,C 180,E1 -11463.871,E2 -11463.871} C_VEL
LIN {X 0,Y 391.633,Z 476.289,A -85,B 0,C 180,E1 -11465.359,E2 -11465.359} C_VEL
LIN {X 0,Y 392.474,Z 467.389,A -85,B 0,C 180,E1 -11466.698,E2 -11466.698} C_VEL
LIN {X 0,Y 393.353,Z 457.204,A -85,B 0,C 180,E1 -11467.941,E2 -11467.941} C_VEL
LIN {X 0,Y 394.168,Z 447.087,A -85,B 0,C 180,E1 -11468.937,E2 -11468.937} C_VEL
LIN {X 0,Y 394.936,Z 435.563,A -85,B 0,C 180,E1 -11469.835,E2 -11469.835} C_VEL
LIN {X 0,Y 395.149,Z 428.07,A -85,B 0,C 180,E1 -11470.311,E2 -11470.311} C_VEL
LIN {X 0,Y 392.229,Z 415.686,A -85,B 0,C 180,E1 -11471.091,E2 -11471.091} C_VEL
LIN {X 0,Y 389.201,Z 405.084,A -85,B 0,C 180,E1 -11471.633,E2 -11471.633} C_VEL
LIN {X 0,Y 389.329,Z 401.642,A -85,B 0,C 180,E1 -11475.25,E2 -11475.25} C_VEL
LIN {X 0,Y 389.367,Z 398.975,A -85,B 0,C 180,E1 -11478.099,E2 -11478.099} C_VEL
LIN {X 0,Y 389.46,Z 396.414,A -85,B 0,C 180,E1 -11480.887,E2 -11480.887} C_VEL
LIN {X 0,Y 389.606,Z 393.319,A -85,B 0,C 180,E1 -11484.262,E2 -11484.262} C_VEL
LIN {X 0,Y 389.709,Z 391.946,A -85,B 0,C 180,E1 -11486.049,E2 -11486.049} C_VEL
LIN {X 0,Y 389.964,Z 391.915,A -85,B 0,C 180,E1 -11488.49,E2 -11488.49} C_VEL
LIN {X 0,Y 390.1,Z 391.895,A -85,B 0,C 180,E1 -11492.069,E2 -11492.069} C_VEL
LIN {X 0,Y 390.067,Z 391.899,A -85,B 0,C 180,E1 -11495.518,E2 -11495.518} C_VEL
LIN {X 0,Y 390.091,Z 391.896,A -85,B 0,C 180,E1 -11498.88,E2 -11498.88} C_VEL
LIN {X 0,Y 390.129,Z 391.889,A -85,B 0,C 180,E1 -11502.692,E2 -11502.692} C_VEL
LIN {X 0,Y 390.175,Z 391.882,A -85,B 0,C 180,E1 -11506.561,E2 -11506.561} C_VEL
LIN {X 0,Y 390.159,Z 391.885,A -85,B 0,C 180,E1 -11509.623,E2 -11509.623} C_VEL
LIN {X 0,Y 390.299,Z 391.866,A -85,B 0,C 180,E1 -11512.759,E2 -11512.759} C_VEL
LIN {X 0,Y 390.215,Z 391.879,A -85,B 0,C 180,E1 -11514.833,E2 -11514.833} C_VEL
LIN {X 0,Y 390.401,Z 391.857,A -85,B 0,C 180,E1 -11517.937,E2 -11517.937} C_VEL
LIN {X 0,Y 390.531,Z 391.839,A -85,B 0,C 180,E1 -11520,E2 -11520} C_VEL
LIN {X 0,Y 390.329,Z 391.865,A -85,B 0,C 180,E1 -11523.096,E2 -11523.096} C_VEL
LIN {X 0,Y 390.298,Z 391.869,A -85,B 0,C 180,E1 -11527.241,E2 -11527.241} C_VEL
LIN {X 0,Y 390.159,Z 391.887,A -85,B 0,C 180,E1 -11530.378,E2 -11530.378} C_VEL
LIN {X 0,Y 390.15,Z 391.887,A -85,B 0,C 180,E1 -11533.543,E2 -11533.543} C_VEL
LIN {X 0,Y 390.129,Z 391.891,A -85,B 0,C 180,E1 -11537.309,E2 -11537.309} C_VEL
LIN {X 0,Y 390.091,Z 391.898,A -85,B 0,C 180,E1 -11541.12,E2 -11541.12} C_VEL
LIN {X 0,Y 390.068,Z 391.9,A -85,B 0,C 180,E1 -11544.482,E2 -11544.482} C_VEL
LIN {X 0,Y 390.1,Z 391.898,A -85,B 0,C 180,E1 -11547.932,E2 -11547.932} C_VEL
LIN {X 0,Y 390.007,Z 391.907,A -85,B 0,C 180,E1 -11551.506,E2 -11551.506} C_VEL
LIN {X 0,Y 390.07,Z 391.898,A -85,B 0,C 180,E1 -11555.209,E2 -11555.209} C_VEL
LIN {X 0,Y 390.081,Z 391.898,A -85,B 0,C 180,E1 -11559.094,E2 -11559.094} C_VEL
LIN {X 0,Y 390.109,Z 391.899,A -85,B 0,C 180,E1 -11562.389,E2 -11562.389} C_VEL
LIN {X 0,Y 390.124,Z 391.967,A -85,B 0,C 180,E1 -11565.144,E2 -11565.144} C_VEL
LIN {X 0,Y 391.012,Z 397.089,A -85,B 0,C 180,E1 -11568.319,E2 -11568.319} C_VEL
LIN {X 0,Y 391.872,Z 401.914,A -85,B 0,C 180,E1 -11571.123,E2 -11571.123} C_VEL
LIN {X 0,Y 392.45,Z 405.618,A -85,B 0,C 180,E1 -11573.14,E2 -11573.14} C_VEL
LIN {X 0,Y 392.23,Z 410.356,A -85,B 0,C 180,E1 -11575.511,E2 -11575.511} C_VEL
LIN {X 0,Y 391.528,Z 416.938,A -85,B 0,C 180,E1 -11578.634,E2 -11578.634} C_VEL
LIN {X 0,Y 390.848,Z 424.612,A -85,B 0,C 180,E1 -11582.13,E2 -11582.13} C_VEL
LIN {X 0,Y 390.366,Z 431.054,A -85,B 0,C 180,E1 -11584.973,E2 -11584.973} C_VEL
LIN {X 0,Y 389.884,Z 438.862,A -85,B 0,C 180,E1 -11588.316,E2 -11588.316} C_VEL
LIN {X 0,Y 389.556,Z 446.265,A -85,B 0,C 180,E1 -11591.394,E2 -11591.394} C_VEL
LIN {X 0,Y 391.792,Z 460.03,A -85,B 0,C 180,E1 -11591.938,E2 -11591.938} C_VEL
LIN {X 0,Y 393.423,Z 472.37,A -85,B 0,C 180,E1 -11592.616,E2 -11592.616} C_VEL
LIN {X 0,Y 394.15,Z 479.385,A -85,B 0,C 180,E1 -11593.085,E2 -11593.085} C_VEL
LIN {X 0,Y 393.29,Z 490.779,A -85,B 0,C 180,E1 -11593.922,E2 -11593.922} C_VEL
LIN {X 0,Y 392.425,Z 501.768,A -85,B 0,C 180,E1 -11594.951,E2 -11594.951} C_VEL
LIN {X 0,Y 391.651,Z 511.467,A -85,B 0,C 180,E1 -11596.082,E2 -11596.082} C_VEL
LIN {X 0,Y 390.787,Z 521.591,A -85,B 0,C 180,E1 -11597.539,E2 -11597.539} C_VEL
LIN {X 0,Y 389.961,Z 530.273,A -85,B 0,C 180,E1 -11599.094,E2 -11599.094} C_VEL
LIN {X 0,Y 389.451,Z 537.233,A -85,B 0,C 180,E1 -11600.655,E2 -11600.655} C_VEL
LIN {X 0,Y 389.076,Z 542.82,A -85,B 0,C 180,E1 -11602.216,E2 -11602.216} C_VEL
LIN {X 0,Y 388.833,Z 547.991,A -85,B 0,C 180,E1 -11604.096,E2 -11604.096} C_VEL
LIN {X 0,Y 388.729,Z 551.432,A -85,B 0,C 180,E1 -11605.855,E2 -11605.855} C_VEL
LIN {X 0,Y 388.788,Z 553.874,A -85,B 0,C 180,E1 -11607.93,E2 -11607.93} C_VEL
LIN {X 0,Y 388.743,Z 554.495,A -85,B 0,C 180,E1 -11608.966,E2 -11608.966} C_VEL
LIN {X 0,Y 388.743,Z 554.719,A -85,B 0,C 180,E1 -11610.002,E2 -11610.002} C_VEL
LIN {X 0,Y 388.789,Z 553.898,A -85,B 0,C 180,E1 -11612.074,E2 -11612.074} C_VEL
LIN {X 0,Y 388.717,Z 552.891,A -85,B 0,C 180,E1 -11613.111,E2 -11613.111} C_VEL
LIN {X 0,Y 388.73,Z 551.48,A -85,B 0,C 180,E1 -11614.149,E2 -11614.149} C_VEL
LIN {X 0,Y 388.832,Z 548.064,A -85,B 0,C 180,E1 -11615.902,E2 -11615.902} C_VEL
LIN {X 0,Y 389.08,Z 542.899,A -85,B 0,C 180,E1 -11617.788,E2 -11617.788} C_VEL
LIN {X 0,Y 389.455,Z 537.324,A -85,B 0,C 180,E1 -11619.349,E2 -11619.349} C_VEL
LIN {X 0,Y 389.961,Z 530.367,A -85,B 0,C 180,E1 -11620.91,E2 -11620.91} C_VEL
LIN {X 0,Y 390.809,Z 521.668,A -85,B 0,C 180,E1 -11622.464,E2 -11622.464} C_VEL
LIN {X 0,Y 391.664,Z 511.525,A -85,B 0,C 180,E1 -11623.921,E2 -11623.921} C_VEL
LIN {X 0,Y 392.408,Z 501.78,A -85,B 0,C 180,E1 -11625.054,E2 -11625.054} C_VEL
LIN {X 0,Y 393.333,Z 490.707,A -85,B 0,C 180,E1 -11626.08,E2 -11626.08} C_VEL
LIN {X 0,Y 394.165,Z 479.293,A -85,B 0,C 180,E1 -11626.912,E2 -11626.912} C_VEL
LIN {X 0,Y 392.669,Z 466.393,A -85,B 0,C 180,E1 -11627.716,E2 -11627.716} C_VEL
LIN {X 0,Y 390.587,Z 452.822,A -85,B 0,C 180,E1 -11628.342,E2 -11628.342} C_VEL
LIN {X 0,Y 389.568,Z 446.658,A -85,B 0,C 180,E1 -11628.576,E2 -11628.576} C_VEL
LIN {X 0,Y 389.955,Z 439.264,A -85,B 0,C 180,E1 -11631.684,E2 -11631.684} C_VEL
LIN {X 0,Y 390.406,Z 431.451,A -85,B 0,C 180,E1 -11635.028,E2 -11635.028} C_VEL
LIN {X 0,Y 390.969,Z 424.098,A -85,B 0,C 180,E1 -11638.258,E2 -11638.258} C_VEL
LIN {X 0,Y 391.729,Z 415.996,A -85,B 0,C 180,E1 -11641.945,E2 -11641.945} C_VEL
LIN {X 0,Y 392.36,Z 409.571,A -85,B 0,C 180,E1 -11644.974,E2 -11644.974} C_VEL
LIN {X 0,Y 392.464,Z 405.733,A -85,B 0,C 180,E1 -11646.863,E2 -11646.863} C_VEL
LIN {X 0,Y 391.666,Z 400.749,A -85,B 0,C 180,E1 -11649.503,E2 -11649.503} C_VEL
LIN {X 0,Y 390.512,Z 394.276,A -85,B 0,C 180,E1 -11653.149,E2 -11653.149} C_VEL
LIN {X 0,Y 390.06,Z 391.9,A -85,B 0,C 180,E1 -11654.645,E2 -11654.645} C_VEL
LIN {X 0,Y 390.037,Z 391.902,A -85,B 0,C 180,E1 -11658.187,E2 -11658.187} C_VEL
LIN {X 0,Y 390.094,Z 391.896,A -85,B 0,C 180,E1 -11660.908,E2 -11660.908} C_VEL
LIN {X 0,Y 390.091,Z 391.897,A -85,B 0,C 180,E1 -11664.793,E2 -11664.793} C_VEL
LIN {X 0,Y 390.03,Z 391.904,A -85,B 0,C 180,E1 -11668.496,E2 -11668.496} C_VEL
LIN {X 0,Y 390.124,Z 391.889,A -85,B 0,C 180,E1 -11672.07,E2 -11672.07} C_VEL
LIN {X 0,Y 390.086,Z 391.892,A -85,B 0,C 180,E1 -11675.52,E2 -11675.52} C_VEL
LIN {X 0,Y 390.062,Z 391.898,A -85,B 0,C 180,E1 -11678.878,E2 -11678.878} C_VEL
LIN {X 0,Y 390.134,Z 391.89,A -85,B 0,C 180,E1 -11682.167,E2 -11682.167} C_VEL
LIN {X 0,Y 390.15,Z 391.884,A -85,B 0,C 180,E1 -11685.393,E2 -11685.393} C_VEL
LIN {X 0,Y 390.154,Z 391.887,A -85,B 0,C 180,E1 -11688.571,E2 -11688.571} C_VEL
LIN {X 0,Y 390.313,Z 391.868,A -85,B 0,C 180,E1 -11692.032,E2 -11692.032} C_VEL
LIN {X 0,Y 390.229,Z 391.875,A -85,B 0,C 180,E1 -11694.833,E2 -11694.833} C_VEL
LIN {X 0,Y 390.423,Z 391.854,A -85,B 0,C 180,E1 -11697.937,E2 -11697.937} C_VEL
LIN {X 0,Y 390.553,Z 391.839,A -85,B 0,C 180,E1 -11700,E2 -11700} C_VEL
LIN {X 0,Y 390.314,Z 391.864,A -85,B 0,C 180,E1 -11703.096,E2 -11703.096} C_VEL
LIN {X 0,Y 390.312,Z 391.864,A -85,B 0,C 180,E1 -11706.672,E2 -11706.672} C_VEL
LIN {X 0,Y 390.211,Z 391.878,A -85,B 0,C 180,E1 -11709.329,E2 -11709.329} C_VEL
LIN {X 0,Y 390.201,Z 391.88,A -85,B 0,C 180,E1 -11713.438,E2 -11713.438} C_VEL
LIN {X 0,Y 390.155,Z 391.886,A -85,B 0,C 180,E1 -11717.307,E2 -11717.307} C_VEL
LIN {X 0,Y 390.093,Z 391.892,A -85,B 0,C 180,E1 -11720.47,E2 -11720.47} C_VEL
LIN {X 0,Y 390.095,Z 391.895,A -85,B 0,C 180,E1 -11723.35,E2 -11723.35} C_VEL
LIN {X 0,Y 390.119,Z 391.888,A -85,B 0,C 180,E1 -11726.768,E2 -11726.768} C_VEL
LIN {X 0,Y 390.045,Z 391.897,A -85,B 0,C 180,E1 -11730.299,E2 -11730.299} C_VEL
LIN {X 0,Y 390.074,Z 391.895,A -85,B 0,C 180,E1 -11734.024,E2 -11734.024} C_VEL
LIN {X 0,Y 390.049,Z 391.901,A -85,B 0,C 180,E1 -11737.55,E2 -11737.55} C_VEL
LIN {X 0,Y 390.062,Z 391.897,A -85,B 0,C 180,E1 -11740.821,E2 -11740.821} C_VEL
LIN {X 0,Y 390.06,Z 391.896,A -85,B 0,C 180,E1 -11743.885,E2 -11743.885} C_VEL
LIN {X 0,Y 390.062,Z 391.897,A -85,B 0,C 180,E1 -11746.789,E2 -11746.789} C_VEL
LIN {X 0,Y 390.062,Z 391.897,A -85,B 0,C 180,E1 -11749.56,E2 -11749.56} C_VEL
LIN {X 0,Y 390.049,Z 391.898,A -85,B 0,C 180,E1 -11752.448,E2 -11752.448} C_VEL
LIN {X 0,Y 390.074,Z 391.894,A -85,B 0,C 180,E1 -11756.044,E2 -11756.044} C_VEL
LIN {X 0,Y 390.052,Z 391.896,A -85,B 0,C 180,E1 -11759.868,E2 -11759.868} C_VEL
LIN {X 0,Y 390.119,Z 391.89,A -85,B 0,C 180,E1 -11763.231,E2 -11763.231} C_VEL
LIN {X 0,Y 390.112,Z 391.894,A -85,B 0,C 180,E1 -11766.749,E2 -11766.749} C_VEL
LIN {X 0,Y 390.109,Z 391.89,A -85,B 0,C 180,E1 -11769.982,E2 -11769.982} C_VEL
LIN {X 0,Y 390.143,Z 391.886,A -85,B 0,C 180,E1 -11773.247,E2 -11773.247} C_VEL
LIN {X 0,Y 390.157,Z 391.888,A -85,B 0,C 180,E1 -11776.585,E2 -11776.585} C_VEL
LIN {X 0,Y 389.917,Z 391.914,A -85,B 0,C 180,E1 -11779.614,E2 -11779.614} C_VEL
LIN {X 0,Y 389.689,Z 391.947,A -85,B 0,C 180,E1 -11781.703,E2 -11781.703} C_VEL
LIN {X 0,Y 389.607,Z 393.61,A -85,B 0,C 180,E1 -11783.785,E2 -11783.785} C_VEL
LIN {X 0,Y 389.646,Z 395.574,A -85,B 0,C 180,E1 -11785.861,E2 -11785.861} C_VEL
LIN {X 0,Y 389.223,Z 399.582,A -85,B 0,C 180,E1 -11789.998,E2 -11789.998} C_VEL
LIN {X 0,Y 389.345,Z 402.666,A -85,B 0,C 180,E1 -11793.102,E2 -11793.102} C_VEL
LIN {X 0,Y 389.304,Z 404.353,A -85,B 0,C 180,E1 -11794.625,E2 -11794.625} C_VEL
LIN {X 0,Y 392.75,Z 417.23,A -85,B 0,C 180,E1 -11795.26,E2 -11795.26} C_VEL
LIN {X 0,Y 394.846,Z 427.19,A -85,B 0,C 180,E1 -11795.872,E2 -11795.872} C_VEL
LIN {X 0,Y 394.893,Z 431.325,A -85,B 0,C 180,E1 -11796.128,E2 -11796.128} C_VEL
LIN {X 0,Y 394.105,Z 443.922,A -85,B 0,C 180,E1 -11797.04,E2 -11797.04} C_VEL
LIN {X 0,Y 393.383,Z 453.848,A -85,B 0,C 180,E1 -11797.956,E2 -11797.956} C_VEL
LIN {X 0,Y 392.492,Z 464.25,A -85,B 0,C 180,E1 -11799.142,E2 -11799.142} C_VEL
LIN {X 0,Y 391.727,Z 472.735,A -85,B 0,C 180,E1 -11800.333,E2 -11800.333} C_VEL
LIN {X 0,Y 390.892,Z 481.939,A -85,B 0,C 180,E1 -11801.93,E2 -11801.93} C_VEL
LIN {X 0,Y 390.229,Z 489.337,A -85,B 0,C 180,E1 -11803.538,E2 -11803.538} C_VEL
LIN {X 0,Y 389.721,Z 495.201,A -85,B 0,C 180,E1 -11805.156,E2 -11805.156} C_VEL
LIN {X 0,Y 389.305,Z 500.086,A -85,B 0,C 180,E1 -11806.904,E2 -11806.904} C_VEL
LIN {X 0,Y 389.135,Z 502.23,A -85,B 0,C 180,E1 -11807.878,E2 -11807.878} C_VEL
LIN {X 0,Y 388.894,Z 504.563,A -85,B 0,C 180,E1 -11809.248,E2 -11809.248} C_VEL
LIN {X 0,Y 388.718,Z 506.681,A -85,B 0,C 180,E1 -11811.196,E2 -11811.196} C_VEL
LIN {X 0,Y 388.684,Z 507.336,A -85,B 0,C 180,E1 -11812.756,E2 -11812.756} C_VEL
LIN {X 0,Y 388.68,Z 507.253,A -85,B 0,C 180,E1 -11813.735,E2 -11813.735} C_VEL
LIN {X 0,Y 388.043,Z 507.025,A -85,B 0,C 180,E1 -11814.6,E2 -11814.6} C_VEL
LIN {X 0,Y 385.313,Z 506.099,A -85,B 0,C 180,E1 -11816.007,E2 -11816.007} C_VEL
LIN {X 0,Y 383.06,Z 504.907,A -85,B 0,C 180,E1 -11817.132,E2 -11817.132} C_VEL
LIN {X 0,Y 382.168,Z 503.622,A -85,B 0,C 180,E1 -11817.988,E2 -11817.988} C_VEL
LIN {X 0,Y 382.136,Z 503.091,A -85,B 0,C 180,E1 -11818.274,E2 -11818.274} C_VEL
LIN {X 0,Y 382.415,Z 499.945,A -85,B 0,C 180,E1 -11819.746,E2 -11819.746} C_VEL
LIN {X 0,Y 382.899,Z 494.784,A -85,B 0,C 180,E1 -11821.538,E2 -11821.538} C_VEL
LIN {X 0,Y 383.607,Z 488.013,A -85,B 0,C 180,E1 -11823.338,E2 -11823.338} C_VEL
LIN {X 0,Y 384.296,Z 481.014,A -85,B 0,C 180,E1 -11824.819,E2 -11824.819} C_VEL
LIN {X 0,Y 385.191,Z 472.26,A -85,B 0,C 180,E1 -11826.311,E2 -11826.311} C_VEL
LIN {X 0,Y 386.141,Z 461.868,A -85,B 0,C 180,E1 -11827.73,E2 -11827.73} C_VEL
LIN {X 0,Y 387.018,Z 452.068,A -85,B 0,C 180,E1 -11828.806,E2 -11828.806} C_VEL
LIN {X 0,Y 387.893,Z 441.031,A -85,B 0,C 180,E1 -11829.774,E2 -11829.774} C_VEL
LIN {X 0,Y 388.451,Z 429.849,A -85,B 0,C 180,E1 -11830.546,E2 -11830.546} C_VEL
LIN {X 0,Y 385.594,Z 417.517,A -85,B 0,C 180,E1 -11831.361,E2 -11831.361} C_VEL
LIN {X 0,Y 382.156,Z 405.526,A -85,B 0,C 180,E1 -11832.011,E2 -11832.011} C_VEL
LIN {X 0,Y 382.297,Z 401.963,A -85,B 0,C 180,E1 -11835.8,E2 -11835.8} C_VEL
LIN {X 0,Y 382.331,Z 399.117,A -85,B 0,C 180,E1 -11838.904,E2 -11838.904} C_VEL
LIN {X 0,Y 382.495,Z 395.661,A -85,B 0,C 180,E1 -11842.674,E2 -11842.674} C_VEL
LIN {X 0,Y 382.622,Z 392.974,A -85,B 0,C 180,E1 -11845.742,E2 -11845.742} C_VEL
LIN {X 0,Y 382.9,Z 392.797,A -85,B 0,C 180,E1 -11847.84,E2 -11847.84} C_VEL
LIN {X 0,Y 382.968,Z 392.782,A -85,B 0,C 180,E1 -11850.298,E2 -11850.298} C_VEL
LIN {X 0,Y 383.063,Z 392.772,A -85,B 0,C 180,E1 -11854.019,E2 -11854.019} C_VEL
LIN {X 0,Y 383.04,Z 392.775,A -85,B 0,C 180,E1 -11857.337,E2 -11857.337} C_VEL
LIN {X 0,Y 383.058,Z 392.772,A -85,B 0,C 180,E1 -11860.716,E2 -11860.716} C_VEL
LIN {X 0,Y 383.061,Z 392.769,A -85,B 0,C 180,E1 -11864.026,E2 -11864.026} C_VEL
LIN {X 0,Y 383.122,Z 392.761,A -85,B 0,C 180,E1 -11867.283,E2 -11867.283} C_VEL
LIN {X 0,Y 383.137,Z 392.759,A -85,B 0,C 180,E1 -11870.498,E2 -11870.498} C_VEL
LIN {X 0,Y 383.254,Z 392.744,A -85,B 0,C 180,E1 -11872.625,E2 -11872.625} C_VEL
LIN {X 0,Y 383.187,Z 392.754,A -85,B 0,C 180,E1 -11874.738,E2 -11874.738} C_VEL
LIN {X 0,Y 383.369,Z 392.733,A -85,B 0,C 180,E1 -11877.899,E2 -11877.899} C_VEL
LIN {X 0,Y 383.501,Z 392.715,A -85,B 0,C 180,E1 -11880,E2 -11880} C_VEL
LIN {X 0,Y 383.263,Z 392.745,A -85,B 0,C 180,E1 -11883.154,E2 -11883.154} C_VEL
LIN {X 0,Y 383.267,Z 392.746,A -85,B 0,C 180,E1 -11886.317,E2 -11886.317} C_VEL
LIN {X 0,Y 383.241,Z 392.748,A -85,B 0,C 180,E1 -11888.436,E2 -11888.436} C_VEL
LIN {X 0,Y 383.088,Z 392.769,A -85,B 0,C 180,E1 -11891.642,E2 -11891.642} C_VEL
LIN {X 0,Y 383.092,Z 392.766,A -85,B 0,C 180,E1 -11894.883,E2 -11894.883} C_VEL
LIN {X 0,Y 383.076,Z 392.77,A -85,B 0,C 180,E1 -11898.173,E2 -11898.173} C_VEL
LIN {X 0,Y 383.058,Z 392.772,A -85,B 0,C 180,E1 -11901.527,E2 -11901.527} C_VEL
LIN {X 0,Y 383.038,Z 392.777,A -85,B 0,C 180,E1 -11904.961,E2 -11904.961} C_VEL
LIN {X 0,Y 383,Z 392.781,A -85,B 0,C 180,E1 -11908.496,E2 -11908.496} C_VEL
LIN {X 0,Y 382.993,Z 392.781,A -85,B 0,C 180,E1 -11912.151,E2 -11912.151} C_VEL
LIN {X 0,Y 383.003,Z 392.779,A -85,B 0,C 180,E1 -11914.67,E2 -11914.67} C_VEL
LIN {X 0,Y 382.989,Z 392.78,A -85,B 0,C 180,E1 -11917.906,E2 -11917.906} C_VEL
LIN {X 0,Y 383.033,Z 392.78,A -85,B 0,C 180,E1 -11921.341,E2 -11921.341} C_VEL
LIN {X 0,Y 383.1,Z 392.925,A -85,B 0,C 180,E1 -11924.767,E2 -11924.767} C_VEL
LIN {X 0,Y 383.98,Z 398.04,A -85,B 0,C 180,E1 -11928.036,E2 -11928.036} C_VEL
LIN {X 0,Y 384.869,Z 402.969,A -85,B 0,C 180,E1 -11930.954,E2 -11930.954} C_VEL
LIN {X 0,Y 385.475,Z 407.288,A -85,B 0,C 180,E1 -11933.342,E2 -11933.342} C_VEL
LIN {X 0,Y 385.191,Z 411.635,A -85,B 0,C 180,E1 -11935.559,E2 -11935.559} C_VEL
LIN {X 0,Y 384.349,Z 419.267,A -85,B 0,C 180,E1 -11939.252,E2 -11939.252} C_VEL
LIN {X 0,Y 383.687,Z 426.84,A -85,B 0,C 180,E1 -11942.75,E2 -11942.75} C_VEL
LIN {X 0,Y 383.206,Z 433.286,A -85,B 0,C 180,E1 -11945.631,E2 -11945.631} C_VEL
LIN {X 0,Y 382.665,Z 442.398,A -85,B 0,C 180,E1 -11949.579,E2 -11949.579} C_VEL
LIN {X 0,Y 382.52,Z 445.719,A -85,B 0,C 180,E1 -11951.004,E2 -11951.004} C_VEL
LIN {X 0,Y 384.944,Z 460.542,A -85,B 0,C 180,E1 -11951.639,E2 -11951.639} C_VEL
LIN {X 0,Y 386.678,Z 474.139,A -85,B 0,C 180,E1 -11952.43,E2 -11952.43} C_VEL
LIN {X 0,Y 387.263,Z 480.881,A -85,B 0,C 180,E1 -11952.901,E2 -11952.901} C_VEL
LIN {X 0,Y 386.191,Z 493.36,A -85,B 0,C 180,E1 -11953.89,E2 -11953.89} C_VEL
LIN {X 0,Y 385.17,Z 504.916,A -85,B 0,C 180,E1 -11955.067,E2 -11955.067} C_VEL
LIN {X 0,Y 384.421,Z 514.249,A -85,B 0,C 180,E1 -11956.254,E2 -11956.254} C_VEL
LIN {X 0,Y 383.64,Z 522.772,A -85,B 0,C 180,E1 -11957.572,E2 -11957.572} C_VEL
LIN {X 0,Y 382.838,Z 531.104,A -85,B 0,C 180,E1 -11959.157,E2 -11959.157} C_VEL
LIN {X 0,Y 382.332,Z 537.838,A -85,B 0,C 180,E1 -11960.746,E2 -11960.746} C_VEL
LIN {X 0,Y 381.953,Z 544.01,A -85,B 0,C 180,E1 -11962.602,E2 -11962.602} C_VEL
LIN {X 0,Y 381.734,Z 547.932,A -85,B 0,C 180,E1 -11964.145,E2 -11964.145} C_VEL
LIN {X 0,Y 381.658,Z 551.005,A -85,B 0,C 180,E1 -11965.778,E2 -11965.778} C_VEL
LIN {X 0,Y 381.704,Z 553.444,A -85,B 0,C 180,E1 -11967.892,E2 -11967.892} C_VEL
LIN {X 0,Y 381.676,Z 554.066,A -85,B 0,C 180,E1 -11968.947,E2 -11968.947} C_VEL
LIN {X 0,Y 381.672,Z 554.289,A -85,B 0,C 180,E1 -11970.002,E2 -11970.002} C_VEL
LIN {X 0,Y 381.676,Z 554.073,A -85,B 0,C 180,E1 -11971.057,E2 -11971.057} C_VEL
LIN {X 0,Y 381.704,Z 553.465,A -85,B 0,C 180,E1 -11972.112,E2 -11972.112} C_VEL
LIN {X 0,Y 381.658,Z 551.044,A -85,B 0,C 180,E1 -11974.226,E2 -11974.226} C_VEL
LIN {X 0,Y 381.734,Z 547.991,A -85,B 0,C 180,E1 -11975.854,E2 -11975.854} C_VEL
LIN {X 0,Y 381.93,Z 544.063,A -85,B 0,C 180,E1 -11977.403,E2 -11977.403} C_VEL
LIN {X 0,Y 382.336,Z 537.886,A -85,B 0,C 180,E1 -11979.258,E2 -11979.258} C_VEL
LIN {X 0,Y 382.838,Z 531.147,A -85,B 0,C 180,E1 -11980.848,E2 -11980.848} C_VEL
LIN {X 0,Y 383.661,Z 522.803,A -85,B 0,C 180,E1 -11982.431,E2 -11982.431} C_VEL
LIN {X 0,Y 384.433,Z 514.231,A -85,B 0,C 180,E1 -11983.75,E2 -11983.75} C_VEL
LIN {X 0,Y 385.299,Z 503.653,A -85,B 0,C 180,E1 -11985.067,E2 -11985.067} C_VEL
LIN {X 0,Y 386.211,Z 493.202,A -85,B 0,C 180,E1 -11986.113,E2 -11986.113} C_VEL
LIN {X 0,Y 387.159,Z 482.126,A -85,B 0,C 180,E1 -11986.993,E2 -11986.993} C_VEL
LIN {X 0,Y 387.09,Z 477.45,A -85,B 0,C 180,E1 -11987.318,E2 -11987.318} C_VEL
LIN {X 0,Y 385.58,Z 465.798,A -85,B 0,C 180,E1 -11988.053,E2 -11988.053} C_VEL
LIN {X 0,Y 383.567,Z 452.425,A -85,B 0,C 180,E1 -11988.681,E2 -11988.681} C_VEL
LIN {X 0,Y 382.532,Z 446.237,A -85,B 0,C 180,E1 -11988.93,E2 -11988.93} C_VEL
LIN {X 0,Y 382.917,Z 438.872,A -85,B 0,C 180,E1 -11992.104,E2 -11992.104} C_VEL
LIN {X 0,Y 383.467,Z 431.094,A -85,B 0,C 180,E1 -11995.513,E2 -11995.513} C_VEL
LIN {X 0,Y 384.1,Z 423.35,A -85,B 0,C 180,E1 -11999.009,E2 -11999.009} C_VEL
LIN {X 0,Y 384.835,Z 415.147,A -85,B 0,C 180,E1 -12002.852,E2 -12002.852} C_VEL
LIN {X 0,Y 385.468,Z 409.265,A -85,B 0,C 180,E1 -12005.694,E2 -12005.694} C_VEL
LIN {X 0,Y 385.271,Z 405.504,A -85,B 0,C 180,E1 -12007.641,E2 -12007.641} C_VEL
LIN {X 0,Y 384.171,Z 399.077,A -85,B 0,C 180,E1 -12011.193,E2 -12011.193} C_VEL
LIN {X 0,Y 383.076,Z 393.182,A -85,B 0,C 180,E1 -12014.688,E2 -12014.688} C_VEL
LIN {X 0,Y 383.026,Z 392.777,A -85,B 0,C 180,E1 -12015.052,E2 -12015.052} C_VEL
LIN {X 0,Y 382.99,Z 392.78,A -85,B 0,C 180,E1 -12018.653,E2 -12018.653} C_VEL
LIN {X 0,Y 383.005,Z 392.778,A -85,B 0,C 180,E1 -12022.097,E2 -12022.097} C_VEL
LIN {X 0,Y 383.024,Z 392.773,A -85,B 0,C 180,E1 -12025.332,E2 -12025.332} C_VEL
LIN {X 0,Y 382.989,Z 392.778,A -85,B 0,C 180,E1 -12029.082,E2 -12029.082} C_VEL
LIN {X 0,Y 383.063,Z 392.772,A -85,B 0,C 180,E1 -12032.698,E2 -12032.698} C_VEL
LIN {X 0,Y 383.058,Z 392.769,A -85,B 0,C 180,E1 -12035.04,E2 -12035.04} C_VEL
LIN {X 0,Y 382.999,Z 392.78,A -85,B 0,C 180,E1 -12038.469,E2 -12038.469} C_VEL
LIN {X 0,Y 383.069,Z 392.767,A -85,B 0,C 180,E1 -12041.827,E2 -12041.827} C_VEL
LIN {X 0,Y 383.116,Z 392.761,A -85,B 0,C 180,E1 -12045.118,E2 -12045.118} C_VEL
LIN {X 0,Y 383.103,Z 392.767,A -85,B 0,C 180,E1 -12048.358,E2 -12048.358} C_VEL
LIN {X 0,Y 383.27,Z 392.744,A -85,B 0,C 180,E1 -12051.976,E2 -12051.976} C_VEL
LIN {X 0,Y 383.201,Z 392.751,A -85,B 0,C 180,E1 -12054.738,E2 -12054.738} C_VEL
LIN {X 0,Y 383.39,Z 392.73,A -85,B 0,C 180,E1 -12057.899,E2 -12057.899} C_VEL
LIN {X 0,Y 383.523,Z 392.714,A -85,B 0,C 180,E1 -12060,E2 -12060} C_VEL
LIN {X 0,Y 383.251,Z 392.744,A -85,B 0,C 180,E1 -12063.154,E2 -12063.154} C_VEL
LIN {X 0,Y 383.272,Z 392.741,A -85,B 0,C 180,E1 -12066.667,E2 -12066.667} C_VEL
LIN {X 0,Y 383.266,Z 392.743,A -85,B 0,C 180,E1 -12068.435,E2 -12068.435} C_VEL
LIN {X 0,Y 383.103,Z 392.766,A -85,B 0,C 180,E1 -12071.642,E2 -12071.642} C_VEL
LIN {X 0,Y 383.116,Z 392.76,A -85,B 0,C 180,E1 -12074.881,E2 -12074.881} C_VEL
LIN {X 0,Y 383.069,Z 392.768,A -85,B 0,C 180,E1 -12078.173,E2 -12078.173} C_VEL
LIN {X 0,Y 382.999,Z 392.779,A -85,B 0,C 180,E1 -12081.531,E2 -12081.531} C_VEL
LIN {X 0,Y 383.058,Z 392.768,A -85,B 0,C 180,E1 -12084.96,E2 -12084.96} C_VEL
LIN {X 0,Y 383.035,Z 392.77,A -85,B 0,C 180,E1 -12088.27,E2 -12088.27} C_VEL
LIN {X 0,Y 383.015,Z 392.773,A -85,B 0,C 180,E1 -12092.149,E2 -12092.149} C_VEL
LIN {X 0,Y 383.024,Z 392.772,A -85,B 0,C 180,E1 -12094.667,E2 -12094.667} C_VEL
LIN {X 0,Y 383.005,Z 392.775,A -85,B 0,C 180,E1 -12097.903,E2 -12097.903} C_VEL
LIN {X 0,Y 382.99,Z 392.781,A -85,B 0,C 180,E1 -12101.347,E2 -12101.347} C_VEL
LIN {X 0,Y 383.001,Z 392.774,A -85,B 0,C 180,E1 -12104.302,E2 -12104.302} C_VEL
LIN {X 0,Y 383.016,Z 392.778,A -85,B 0,C 180,E1 -12107.239,E2 -12107.239} C_VEL
LIN {X 0,Y 383.021,Z 392.773,A -85,B 0,C 180,E1 -12110.413,E2 -12110.413} C_VEL
LIN {X 0,Y 383.031,Z 392.771,A -85,B 0,C 180,E1 -12114.043,E2 -12114.043} C_VEL
LIN {X 0,Y 382.992,Z 392.777,A -85,B 0,C 180,E1 -12117.577,E2 -12117.577} C_VEL
LIN {X 0,Y 382.997,Z 392.776,A -85,B 0,C 180,E1 -12120.299,E2 -12120.299} C_VEL
LIN {X 0,Y 383.086,Z 392.764,A -85,B 0,C 180,E1 -12124.019,E2 -12124.019} C_VEL
LIN {X 0,Y 383.013,Z 392.774,A -85,B 0,C 180,E1 -12127.334,E2 -12127.334} C_VEL
LIN {X 0,Y 383.065,Z 392.772,A -85,B 0,C 180,E1 -12130.715,E2 -12130.715} C_VEL
LIN {X 0,Y 383.085,Z 392.765,A -85,B 0,C 180,E1 -12134.025,E2 -12134.025} C_VEL
LIN {X 0,Y 383.075,Z 392.766,A -85,B 0,C 180,E1 -12137.28,E2 -12137.28} C_VEL
LIN {X 0,Y 382.776,Z 392.808,A -85,B 0,C 180,E1 -12140.487,E2 -12140.487} C_VEL
LIN {X 0,Y 382.658,Z 392.821,A -85,B 0,C 180,E1 -12141.549,E2 -12141.549} C_VEL
LIN {X 0,Y 382.62,Z 393.425,A -85,B 0,C 180,E1 -12142.692,E2 -12142.692} C_VEL
LIN {X 0,Y 382.61,Z 396.318,A -85,B 0,C 180,E1 -12145.785,E2 -12145.785} C_VEL
LIN {X 0,Y 382.171,Z 400.436,A -85,B 0,C 180,E1 -12149.998,E2 -12149.998} C_VEL
LIN {X 0,Y 382.3,Z 403.451,A -85,B 0,C 180,E1 -12153.159,E2 -12153.159} C_VEL
LIN {X 0,Y 382.253,Z 404.655,A -85,B 0,C 180,E1 -12154.281,E2 -12154.281} C_VEL
LIN {X 0,Y 385.754,Z 417.82,A -85,B 0,C 180,E1 -12154.946,E2 -12154.946} C_VEL
LIN {X 0,Y 388.207,Z 429.762,A -85,B 0,C 180,E1 -12155.712,E2 -12155.712} C_VEL
LIN {X 0,Y 387.488,Z 441.254,A -85,B 0,C 180,E1 -12156.507,E2 -12156.507} C_VEL
LIN {X 0,Y 386.604,Z 453.062,A -85,B 0,C 180,E1 -12157.571,E2 -12157.571} C_VEL
LIN {X 0,Y 385.698,Z 463.682,A -85,B 0,C 180,E1 -12158.776,E2 -12158.776} C_VEL
LIN {X 0,Y 384.862,Z 472.698,A -85,B 0,C 180,E1 -12160.04,E2 -12160.04} C_VEL
LIN {X 0,Y 383.976,Z 481.721,A -85,B 0,C 180,E1 -12161.613,E2 -12161.613} C_VEL
LIN {X 0,Y 383.331,Z 488.75,A -85,B 0,C 180,E1 -12163.133,E2 -12163.133} C_VEL
LIN {X 0,Y 382.727,Z 495.24,A -85,B 0,C 180,E1 -12164.895,E2 -12164.895} C_VEL
LIN {X 0,Y 382.321,Z 499.835,A -85,B 0,C 180,E1 -12166.512,E2 -12166.512} C_VEL
LIN {X 0,Y 381.991,Z 503.474,A -85,B 0,C 180,E1 -12168.224,E2 -12168.224} C_VEL
LIN {X 0,Y 381.727,Z 506.173,A -85,B 0,C 180,E1 -12170.121,E2 -12170.121} C_VEL
LIN {X 0,Y 381.611,Z 507.384,A -85,B 0,C 180,E1 -12171.61,E2 -12171.61} C_VEL
LIN {X 0,Y 381.605,Z 507.801,A -85,B 0,C 180,E1 -12172.95,E2 -12172.95} C_VEL
LIN {X 0,Y 381.603,Z 507.72,A -85,B 0,C 180,E1 -12173.899,E2 -12173.899} C_VEL
LIN {X 0,Y 381.721,Z 506.792,A -85,B 0,C 180,E1 -12175.557,E2 -12175.557} C_VEL
LIN {X 0,Y 381.967,Z 504.628,A -85,B 0,C 180,E1 -12177.383,E2 -12177.383} C_VEL
LIN {X 0,Y 382.136,Z 503.091,A -85,B 0,C 180,E1 -12178.274,E2 -12178.274} C_VEL
LIN {X 0,Y 381.619,Z 501.454,A -85,B 0,C 180,E1 -12179.122,E2 -12179.122} C_VEL
LIN {X 0,Y 379.028,Z 498.401,A -85,B 0,C 180,E1 -12180.492,E2 -12180.492} C_VEL
LIN {X 0,Y 376.558,Z 494.715,A -85,B 0,C 180,E1 -12181.839,E2 -12181.839} C_VEL
LIN {X 0,Y 376.234,Z 491.999,A -85,B 0,C 180,E1 -12182.638,E2 -12182.638} C_VEL
LIN {X 0,Y 377.007,Z 485.072,A -85,B 0,C 180,E1 -12184.308,E2 -12184.308} C_VEL
LIN {X 0,Y 377.854,Z 477.011,A -85,B 0,C 180,E1 -12185.863,E2 -12185.863} C_VEL
LIN {X 0,Y 378.78,Z 467.819,A -85,B 0,C 180,E1 -12187.287,E2 -12187.287} C_VEL
LIN {X 0,Y 379.705,Z 458.304,A -85,B 0,C 180,E1 -12188.486,E2 -12188.486} C_VEL
LIN {X 0,Y 380.63,Z 447.672,A -85,B 0,C 180,E1 -12189.569,E2 -12189.569} C_VEL
LIN {X 0,Y 381.44,Z 436.604,A -85,B 0,C 180,E1 -12190.46,E2 -12190.46} C_VEL
LIN {X 0,Y 381.624,Z 430.793,A -85,B 0,C 180,E1 -12190.853,E2 -12190.853} C_VEL
LIN {X 0,Y 378.767,Z 418.549,A -85,B 0,C 180,E1 -12191.69,E2 -12191.69} C_VEL
LIN {X 0,Y 375.113,Z 405.961,A -85,B 0,C 180,E1 -12192.41,E2 -12192.41} C_VEL
LIN {X 0,Y 375.238,Z 403.209,A -85,B 0,C 180,E1 -12195.371,E2 -12195.371} C_VEL
LIN {X 0,Y 375.29,Z 399.867,A -85,B 0,C 180,E1 -12199.047,E2 -12199.047} C_VEL
LIN {X 0,Y 375.412,Z 397.357,A -85,B 0,C 180,E1 -12201.845,E2 -12201.845} C_VEL
LIN {X 0,Y 375.571,Z 394.228,A -85,B 0,C 180,E1 -12205.418,E2 -12205.418} C_VEL
LIN {X 0,Y 375.586,Z 393.859,A -85,B 0,C 180,E1 -12205.85,E2 -12205.85} C_VEL
LIN {X 0,Y 375.868,Z 393.671,A -85,B 0,C 180,E1 -12208.43,E2 -12208.43} C_VEL
LIN {X 0,Y 375.964,Z 393.655,A -85,B 0,C 180,E1 -12211.466,E2 -12211.466} C_VEL
LIN {X 0,Y 375.99,Z 393.652,A -85,B 0,C 180,E1 -12214.538,E2 -12214.538} C_VEL
LIN {X 0,Y 376.007,Z 393.65,A -85,B 0,C 180,E1 -12218.048,E2 -12218.048} C_VEL
LIN {X 0,Y 376.013,Z 393.649,A -85,B 0,C 180,E1 -12221.473,E2 -12221.473} C_VEL
LIN {X 0,Y 376.04,Z 393.645,A -85,B 0,C 180,E1 -12224.832,E2 -12224.832} C_VEL
LIN {X 0,Y 376.04,Z 393.645,A -85,B 0,C 180,E1 -12228.136,E2 -12228.136} C_VEL
LIN {X 0,Y 376.238,Z 393.619,A -85,B 0,C 180,E1 -12231.877,E2 -12231.877} C_VEL
LIN {X 0,Y 376.159,Z 393.63,A -85,B 0,C 180,E1 -12234.64,E2 -12234.64} C_VEL
LIN {X 0,Y 376.335,Z 393.609,A -85,B 0,C 180,E1 -12237.86,E2 -12237.86} C_VEL
LIN {X 0,Y 376.47,Z 393.591,A -85,B 0,C 180,E1 -12240,E2 -12240} C_VEL
LIN {X 0,Y 376.199,Z 393.626,A -85,B 0,C 180,E1 -12243.213,E2 -12243.213} C_VEL
LIN {X 0,Y 376.226,Z 393.622,A -85,B 0,C 180,E1 -12246.435,E2 -12246.435} C_VEL
LIN {X 0,Y 376.186,Z 393.627,A -85,B 0,C 180,E1 -12248.596,E2 -12248.596} C_VEL
LIN {X 0,Y 376.04,Z 393.645,A -85,B 0,C 180,E1 -12251.864,E2 -12251.864} C_VEL
LIN {X 0,Y 376.04,Z 393.645,A -85,B 0,C 180,E1 -12255.168,E2 -12255.168} C_VEL
LIN {X 0,Y 376.013,Z 393.649,A -85,B 0,C 180,E1 -12258.527,E2 -12258.527} C_VEL
LIN {X 0,Y 376.007,Z 393.65,A -85,B 0,C 180,E1 -12261.952,E2 -12261.952} C_VEL
LIN {X 0,Y 375.991,Z 393.655,A -85,B 0,C 180,E1 -12265.462,E2 -12265.462} C_VEL
LIN {X 0,Y 375.944,Z 393.661,A -85,B 0,C 180,E1 -12269.082,E2 -12269.082} C_VEL
LIN {X 0,Y 375.933,Z 393.66,A -85,B 0,C 180,E1 -12272.83,E2 -12272.83} C_VEL
LIN {X 0,Y 375.943,Z 393.658,A -85,B 0,C 180,E1 -12275.417,E2 -12275.417} C_VEL
LIN {X 0,Y 375.964,Z 393.656,A -85,B 0,C 180,E1 -12278.273,E2 -12278.273} C_VEL
LIN {X 0,Y 375.977,Z 393.66,A -85,B 0,C 180,E1 -12281.612,E2 -12281.612} C_VEL
LIN {X 0,Y 376.043,Z 393.747,A -85,B 0,C 180,E1 -12284.269,E2 -12284.269} C_VEL
LIN {X 0,Y 376.982,Z 399.172,A -85,B 0,C 180,E1 -12287.849,E2 -12287.849} C_VEL
LIN {X 0,Y 378.006,Z 404.972,A -85,B 0,C 180,E1 -12291.341,E2 -12291.341} C_VEL
LIN {X 0,Y 378.477,Z 408.926,A -85,B 0,C 180,E1 -12293.547,E2 -12293.547} C_VEL
LIN {X 0,Y 378.051,Z 413.879,A -85,B 0,C 180,E1 -12296.106,E2 -12296.106} C_VEL
LIN {X 0,Y 377.231,Z 421.448,A -85,B 0,C 180,E1 -12299.803,E2 -12299.803} C_VEL
LIN {X 0,Y 376.499,Z 429.631,A -85,B 0,C 180,E1 -12303.638,E2 -12303.638} C_VEL
LIN {X 0,Y 375.856,Z 438.086,A -85,B 0,C 180,E1 -12307.463,E2 -12307.463} C_VEL
LIN {X 0,Y 375.493,Z 445.317,A -85,B 0,C 180,E1 -12310.639,E2 -12310.639} C_VEL
LIN {X 0,Y 377.85,Z 459.212,A -85,B 0,C 180,E1 -12311.229,E2 -12311.229} C_VEL
LIN {X 0,Y 379.508,Z 472.525,A -85,B 0,C 180,E1 -12312.005,E2 -12312.005} C_VEL
LIN {X 0,Y 380.397,Z 480.687,A -85,B 0,C 180,E1 -12312.592,E2 -12312.592} C_VEL
LIN {X 0,Y 379.372,Z 493,A -85,B 0,C 180,E1 -12313.592,E2 -12313.592} C_VEL
LIN {X 0,Y 378.291,Z 504.53,A -85,B 0,C 180,E1 -12314.789,E2 -12314.789} C_VEL
LIN {X 0,Y 377.504,Z 513.846,A -85,B 0,C 180,E1 -12315.997,E2 -12315.997} C_VEL
LIN {X 0,Y 376.687,Z 522.362,A -85,B 0,C 180,E1 -12317.339,E2 -12317.339} C_VEL
LIN {X 0,Y 375.827,Z 530.689,A -85,B 0,C 180,E1 -12318.952,E2 -12318.952} C_VEL
LIN {X 0,Y 375.284,Z 537.42,A -85,B 0,C 180,E1 -12320.571,E2 -12320.571} C_VEL
LIN {X 0,Y 374.879,Z 543.587,A -85,B 0,C 180,E1 -12322.461,E2 -12322.461} C_VEL
LIN {X 0,Y 374.699,Z 546.9,A -85,B 0,C 180,E1 -12323.769,E2 -12323.769} C_VEL
LIN {X 0,Y 374.588,Z 550.58,A -85,B 0,C 180,E1 -12325.698,E2 -12325.698} C_VEL
LIN {X 0,Y 374.606,Z 553.016,A -85,B 0,C 180,E1 -12327.852,E2 -12327.852} C_VEL
LIN {X 0,Y 374.61,Z 553.639,A -85,B 0,C 180,E1 -12328.927,E2 -12328.927} C_VEL
LIN {X 0,Y 374.604,Z 553.859,A -85,B 0,C 180,E1 -12330.002,E2 -12330.002} C_VEL
LIN {X 0,Y 374.611,Z 553.641,A -85,B 0,C 180,E1 -12331.077,E2 -12331.077} C_VEL
LIN {X 0,Y 374.622,Z 553.03,A -85,B 0,C 180,E1 -12332.152,E2 -12332.152} C_VEL
LIN {X 0,Y 374.589,Z 550.605,A -85,B 0,C 180,E1 -12334.306,E2 -12334.306} C_VEL
LIN {X 0,Y 374.701,Z 546.926,A -85,B 0,C 180,E1 -12336.234,E2 -12336.234} C_VEL
LIN {X 0,Y 374.946,Z 541.999,A -85,B 0,C 180,E1 -12338.083,E2 -12338.083} C_VEL
LIN {X 0,Y 375.399,Z 536.414,A -85,B 0,C 180,E1 -12339.702,E2 -12339.702} C_VEL
LIN {X 0,Y 375.953,Z 529.441,A -85,B 0,C 180,E1 -12341.322,E2 -12341.322} C_VEL
LIN {X 0,Y 376.868,Z 520.72,A -85,B 0,C 180,E1 -12342.933,E2 -12342.933} C_VEL
LIN {X 0,Y 377.725,Z 511.403,A -85,B 0,C 180,E1 -12344.328,E2 -12344.328} C_VEL
LIN {X 0,Y 378.528,Z 501.983,A -85,B 0,C 180,E1 -12345.481,E2 -12345.481} C_VEL
LIN {X 0,Y 379.513,Z 491.254,A -85,B 0,C 180,E1 -12346.544,E2 -12346.544} C_VEL
LIN {X 0,Y 380.374,Z 480.259,A -85,B 0,C 180,E1 -12347.403,E2 -12347.403} C_VEL
LIN {X 0,Y 378.818,Z 467.352,A -85,B 0,C 180,E1 -12348.273,E2 -12348.273} C_VEL
LIN {X 0,Y 376.908,Z 454.072,A -85,B 0,C 180,E1 -12348.948,E2 -12348.948} C_VEL
LIN {X 0,Y 375.488,Z 445.899,A -85,B 0,C 180,E1 -12349.26,E2 -12349.26} C_VEL
LIN {X 0,Y 375.908,Z 438.469,A -85,B 0,C 180,E1 -12352.538,E2 -12352.538} C_VEL
LIN {X 0,Y 376.562,Z 429.925,A -85,B 0,C 180,E1 -12356.381,E2 -12356.381} C_VEL
LIN {X 0,Y 377.262,Z 421.739,A -85,B 0,C 180,E1 -12360.199,E2 -12360.199} C_VEL
LIN {X 0,Y 377.874,Z 415.541,A -85,B 0,C 180,E1 -12363.181,E2 -12363.181} C_VEL
LIN {X 0,Y 378.471,Z 410.266,A -85,B 0,C 180,E1 -12365.8,E2 -12365.8} C_VEL
LIN {X 0,Y 378.247,Z 406.419,A -85,B 0,C 180,E1 -12367.82,E2 -12367.82} C_VEL
LIN {X 0,Y 377.356,Z 401.329,A -85,B 0,C 180,E1 -12370.683,E2 -12370.683} C_VEL
LIN {X 0,Y 376.454,Z 396.251,A -85,B 0,C 180,E1 -12373.691,E2 -12373.691} C_VEL
LIN {X 0,Y 375.964,Z 393.655,A -85,B 0,C 180,E1 -12375.35,E2 -12375.35} C_VEL
LIN {X 0,Y 375.946,Z 393.658,A -85,B 0,C 180,E1 -12379.134,E2 -12379.134} C_VEL
LIN {X 0,Y 375.969,Z 393.655,A -85,B 0,C 180,E1 -12381.912,E2 -12381.912} C_VEL
LIN {X 0,Y 375.986,Z 393.649,A -85,B 0,C 180,E1 -12385.333,E2 -12385.333} C_VEL
LIN {X 0,Y 375.964,Z 393.655,A -85,B 0,C 180,E1 -12388.438,E2 -12388.438} C_VEL
LIN {X 0,Y 375.99,Z 393.649,A -85,B 0,C 180,E1 -12392.141,E2 -12392.141} C_VEL
LIN {X 0,Y 376.013,Z 393.65,A -85,B 0,C 180,E1 -12394.539,E2 -12394.539} C_VEL
LIN {X 0,Y 375.969,Z 393.652,A -85,B 0,C 180,E1 -12398.046,E2 -12398.046} C_VEL
LIN {X 0,Y 376.015,Z 393.645,A -85,B 0,C 180,E1 -12401.473,E2 -12401.473} C_VEL
LIN {X 0,Y 376.064,Z 393.64,A -85,B 0,C 180,E1 -12404.833,E2 -12404.833} C_VEL
LIN {X 0,Y 376.056,Z 393.644,A -85,B 0,C 180,E1 -12408.137,E2 -12408.137} C_VEL
LIN {X 0,Y 376.225,Z 393.621,A -85,B 0,C 180,E1 -12411.92,E2 -12411.92} C_VEL
LIN {X 0,Y 376.174,Z 393.627,A -85,B 0,C 180,E1 -12414.64,E2 -12414.64} C_VEL
LIN {X 0,Y 376.356,Z 393.606,A -85,B 0,C 180,E1 -12417.86,E2 -12417.86} C_VEL
LIN {X 0,Y 376.492,Z 393.59,A -85,B 0,C 180,E1 -12420,E2 -12420} C_VEL
LIN {X 0,Y 376.189,Z 393.623,A -85,B 0,C 180,E1 -12423.213,E2 -12423.213} C_VEL
LIN {X 0,Y 376.236,Z 393.617,A -85,B 0,C 180,E1 -12426.659,E2 -12426.659} C_VEL
LIN {X 0,Y 376.212,Z 393.62,A -85,B 0,C 180,E1 -12428.595,E2 -12428.595} C_VEL
LIN {X 0,Y 376.056,Z 393.645,A -85,B 0,C 180,E1 -12431.863,E2 -12431.863} C_VEL
LIN {X 0,Y 376.064,Z 393.639,A -85,B 0,C 180,E1 -12435.167,E2 -12435.167} C_VEL
LIN {X 0,Y 376.015,Z 393.645,A -85,B 0,C 180,E1 -12438.526,E2 -12438.526} C_VEL
LIN {X 0,Y 375.969,Z 393.654,A -85,B 0,C 180,E1 -12441.954,E2 -12441.954} C_VEL
LIN {X 0,Y 376.013,Z 393.65,A -85,B 0,C 180,E1 -12445.461,E2 -12445.461} C_VEL
LIN {X 0,Y 375.967,Z 393.652,A -85,B 0,C 180,E1 -12449.079,E2 -12449.079} C_VEL
LIN {X 0,Y 375.955,Z 393.653,A -85,B 0,C 180,E1 -12452.828,E2 -12452.828} C_VEL
LIN {X 0,Y 375.963,Z 393.656,A -85,B 0,C 180,E1 -12455.415,E2 -12455.415} C_VEL
LIN {X 0,Y 375.979,Z 393.649,A -85,B 0,C 180,E1 -12458.27,E2 -12458.27} C_VEL
LIN {X 0,Y 375.94,Z 393.657,A -85,B 0,C 180,E1 -12461.6,E2 -12461.6} C_VEL
LIN {X 0,Y 375.958,Z 393.657,A -85,B 0,C 180,E1 -12465.264,E2 -12465.264} C_VEL
LIN {X 0,Y 375.946,Z 393.658,A -85,B 0,C 180,E1 -12469.132,E2 -12469.132} C_VEL
LIN {X 0,Y 375.97,Z 393.65,A -85,B 0,C 180,E1 -12471.911,E2 -12471.911} C_VEL
LIN {X 0,Y 375.985,Z 393.651,A -85,B 0,C 180,E1 -12475.332,E2 -12475.332} C_VEL
LIN {X 0,Y 375.963,Z 393.653,A -85,B 0,C 180,E1 -12478.437,E2 -12478.437} C_VEL
LIN {X 0,Y 375.988,Z 393.648,A -85,B 0,C 180,E1 -12482.139,E2 -12482.139} C_VEL
LIN {X 0,Y 376.012,Z 393.648,A -85,B 0,C 180,E1 -12484.538,E2 -12484.538} C_VEL
LIN {X 0,Y 375.968,Z 393.651,A -85,B 0,C 180,E1 -12488.044,E2 -12488.044} C_VEL
LIN {X 0,Y 376.014,Z 393.645,A -85,B 0,C 180,E1 -12491.472,E2 -12491.472} C_VEL
LIN {X 0,Y 376.06,Z 393.643,A -85,B 0,C 180,E1 -12494.831,E2 -12494.831} C_VEL
LIN {X 0,Y 376.057,Z 393.641,A -85,B 0,C 180,E1 -12497.039,E2 -12497.039} C_VEL
LIN {X 0,Y 375.752,Z 393.682,A -85,B 0,C 180,E1 -12500.307,E2 -12500.307} C_VEL
LIN {X 0,Y 375.584,Z 394.081,A -85,B 0,C 180,E1 -12502.472,E2 -12502.472} C_VEL
LIN {X 0,Y 375.575,Z 397.071,A -85,B 0,C 180,E1 -12505.705,E2 -12505.705} C_VEL
LIN {X 0,Y 375.111,Z 401.223,A -85,B 0,C 180,E1 -12509.998,E2 -12509.998} C_VEL
LIN {X 0,Y 375.227,Z 404.992,A -85,B 0,C 180,E1 -12513.925,E2 -12513.925} C_VEL
LIN {X 0,Y 378.919,Z 418.922,A -85,B 0,C 180,E1 -12514.652,E2 -12514.652} C_VEL
LIN {X 0,Y 381.409,Z 430.829,A -85,B 0,C 180,E1 -12515.446,E2 -12515.446} C_VEL
LIN {X 0,Y 380.663,Z 442.028,A -85,B 0,C 180,E1 -12516.245,E2 -12516.245} C_VEL
LIN {X 0,Y 379.768,Z 453.565,A -85,B 0,C 180,E1 -12517.307,E2 -12517.307} C_VEL
LIN {X 0,Y 378.795,Z 464.189,A -85,B 0,C 180,E1 -12518.534,E2 -12518.534} C_VEL
LIN {X 0,Y 377.9,Z 473.526,A -85,B 0,C 180,E1 -12519.876,E2 -12519.876} C_VEL
LIN {X 0,Y 377.065,Z 481.506,A -85,B 0,C 180,E1 -12521.284,E2 -12521.284} C_VEL
LIN {X 0,Y 376.349,Z 489.124,A -85,B 0,C 180,E1 -12522.947,E2 -12522.947} C_VEL
LIN {X 0,Y 375.729,Z 495.247,A -85,B 0,C 180,E1 -12524.624,E2 -12524.624} C_VEL
LIN {X 0,Y 375.297,Z 500.048,A -85,B 0,C 180,E1 -12526.311,E2 -12526.311} C_VEL
LIN {X 0,Y 374.946,Z 503.684,A -85,B 0,C 180,E1 -12528.013,E2 -12528.013} C_VEL
LIN {X 0,Y 374.639,Z 506.824,A -85,B 0,C 180,E1 -12530.287,E2 -12530.287} C_VEL
LIN {X 0,Y 374.512,Z 508.024,A -85,B 0,C 180,E1 -12532.041,E2 -12532.041} C_VEL
LIN {X 0,Y 374.511,Z 508.246,A -85,B 0,C 180,E1 -12533.206,E2 -12533.206} C_VEL
LIN {X 0,Y 374.555,Z 507.977,A -85,B 0,C 180,E1 -12534.378,E2 -12534.378} C_VEL
LIN {X 0,Y 374.678,Z 507.068,A -85,B 0,C 180,E1 -12535.795,E2 -12535.795} C_VEL
LIN {X 0,Y 374.993,Z 504.317,A -85,B 0,C 180,E1 -12537.937,E2 -12537.937} C_VEL
LIN {X 0,Y 375.345,Z 500.7,A -85,B 0,C 180,E1 -12539.745,E2 -12539.745} C_VEL
LIN {X 0,Y 375.86,Z 495.683,A -85,B 0,C 180,E1 -12541.568,E2 -12541.568} C_VEL
LIN {X 0,Y 376.234,Z 491.999,A -85,B 0,C 180,E1 -12542.638,E2 -12542.638} C_VEL
LIN {X 0,Y 375.944,Z 489.086,A -85,B 0,C 180,E1 -12543.419,E2 -12543.419} C_VEL
LIN {X 0,Y 373.69,Z 484.074,A -85,B 0,C 180,E1 -12544.68,E2 -12544.68} C_VEL
LIN {X 0,Y 371.484,Z 478.514,A -85,B 0,C 180,E1 -12545.896,E2 -12545.896} C_VEL
LIN {X 0,Y 371.275,Z 474.653,A -85,B 0,C 180,E1 -12546.594,E2 -12546.594} C_VEL
LIN {X 0,Y 372.292,Z 464.672,A -85,B 0,C 180,E1 -12548.061,E2 -12548.061} C_VEL
LIN {X 0,Y 373.32,Z 454.481,A -85,B 0,C 180,E1 -12549.258,E2 -12549.258} C_VEL
LIN {X 0,Y 374.191,Z 444.472,A -85,B 0,C 180,E1 -12550.209,E2 -12550.209} C_VEL
LIN {X 0,Y 374.961,Z 432.591,A -85,B 0,C 180,E1 -12551.105,E2 -12551.105} C_VEL
LIN {X 0,Y 372.172,Z 420.576,A -85,B 0,C 180,E1 -12551.97,E2 -12551.97} C_VEL
LIN {X 0,Y 368.62,Z 408.608,A -85,B 0,C 180,E1 -12552.675,E2 -12552.675} C_VEL
LIN {X 0,Y 368.082,Z 406.44,A -85,B 0,C 180,E1 -12552.786,E2 -12552.786} C_VEL
LIN {X 0,Y 368.166,Z 404.349,A -85,B 0,C 180,E1 -12555.065,E2 -12555.065} C_VEL
LIN {X 0,Y 368.223,Z 401.623,A -85,B 0,C 180,E1 -12558.1,E2 -12558.1} C_VEL
LIN {X 0,Y 368.356,Z 398.637,A -85,B 0,C 180,E1 -12561.463,E2 -12561.463} C_VEL
LIN {X 0,Y 368.506,Z 395.486,A -85,B 0,C 180,E1 -12565.1,E2 -12565.1} C_VEL
LIN {X 0,Y 368.575,Z 394.58,A -85,B 0,C 180,E1 -12566.429,E2 -12566.429} C_VEL
LIN {X 0,Y 368.841,Z 394.545,A -85,B 0,C 180,E1 -12569.038,E2 -12569.038} C_VEL
LIN {X 0,Y 368.943,Z 394.529,A -85,B 0,C 180,E1 -12571.561,E2 -12571.561} C_VEL
LIN {X 0,Y 368.983,Z 394.526,A -85,B 0,C 180,E1 -12574.019,E2 -12574.019} C_VEL
LIN {X 0,Y 368.96,Z 394.528,A -85,B 0,C 180,E1 -12577.607,E2 -12577.607} C_VEL
LIN {X 0,Y 368.974,Z 394.525,A -85,B 0,C 180,E1 -12581.107,E2 -12581.107} C_VEL
LIN {X 0,Y 368.979,Z 394.523,A -85,B 0,C 180,E1 -12584.534,E2 -12584.534} C_VEL
LIN {X 0,Y 368.994,Z 394.522,A -85,B 0,C 180,E1 -12587.906,E2 -12587.906} C_VEL
LIN {X 0,Y 369.21,Z 394.495,A -85,B 0,C 180,E1 -12591.8,E2 -12591.8} C_VEL
LIN {X 0,Y 369.132,Z 394.505,A -85,B 0,C 180,E1 -12594.537,E2 -12594.537} C_VEL
LIN {X 0,Y 369.3,Z 394.485,A -85,B 0,C 180,E1 -12597.819,E2 -12597.819} C_VEL
LIN {X 0,Y 369.44,Z 394.467,A -85,B 0,C 180,E1 -12600,E2 -12600} C_VEL
LIN {X 0,Y 369.305,Z 394.484,A -85,B 0,C 180,E1 -12602.181,E2 -12602.181} C_VEL
LIN {X 0,Y 369.188,Z 394.498,A -85,B 0,C 180,E1 -12606.559,E2 -12606.559} C_VEL
LIN {X 0,Y 369.119,Z 394.508,A -85,B 0,C 180,E1 -12608.761,E2 -12608.761} C_VEL
LIN {X 0,Y 368.994,Z 394.522,A -85,B 0,C 180,E1 -12612.094,E2 -12612.094} C_VEL
LIN {X 0,Y 368.979,Z 394.526,A -85,B 0,C 180,E1 -12615.466,E2 -12615.466} C_VEL
LIN {X 0,Y 368.975,Z 394.525,A -85,B 0,C 180,E1 -12618.893,E2 -12618.893} C_VEL
LIN {X 0,Y 368.961,Z 394.53,A -85,B 0,C 180,E1 -12622.393,E2 -12622.393} C_VEL
LIN {X 0,Y 368.983,Z 394.527,A -85,B 0,C 180,E1 -12625.982,E2 -12625.982} C_VEL
LIN {X 0,Y 368.898,Z 394.537,A -85,B 0,C 180,E1 -12629.692,E2 -12629.692} C_VEL
LIN {X 0,Y 368.881,Z 394.539,A -85,B 0,C 180,E1 -12633.045,E2 -12633.045} C_VEL
LIN {X 0,Y 368.904,Z 394.535,A -85,B 0,C 180,E1 -12636.199,E2 -12636.199} C_VEL
LIN {X 0,Y 368.895,Z 394.538,A -85,B 0,C 180,E1 -12638.954,E2 -12638.954} C_VEL
LIN {X 0,Y 368.929,Z 394.537,A -85,B 0,C 180,E1 -12642.022,E2 -12642.022} C_VEL
LIN {X 0,Y 368.976,Z 394.716,A -85,B 0,C 180,E1 -12643.852,E2 -12643.852} C_VEL
LIN {X 0,Y 369.748,Z 399.036,A -85,B 0,C 180,E1 -12646.826,E2 -12646.826} C_VEL
LIN {X 0,Y 370.622,Z 403.837,A -85,B 0,C 180,E1 -12649.858,E2 -12649.858} C_VEL
LIN {X 0,Y 371.425,Z 408.705,A -85,B 0,C 180,E1 -12652.739,E2 -12652.739} C_VEL
LIN {X 0,Y 371.381,Z 411.878,A -85,B 0,C 180,E1 -12654.462,E2 -12654.462} C_VEL
LIN {X 0,Y 370.712,Z 417.374,A -85,B 0,C 180,E1 -12657.299,E2 -12657.299} C_VEL
LIN {X 0,Y 369.963,Z 424.694,A -85,B 0,C 180,E1 -12660.908,E2 -12660.908} C_VEL
LIN {X 0,Y 369.255,Z 432.583,A -85,B 0,C 180,E1 -12664.647,E2 -12664.647} C_VEL
LIN {X 0,Y 368.615,Z 441.584,A -85,B 0,C 180,E1 -12668.764,E2 -12668.764} C_VEL
LIN {X 0,Y 368.452,Z 444.981,A -85,B 0,C 180,E1 -12670.247,E2 -12670.247} C_VEL
LIN {X 0,Y 370.899,Z 458.738,A -85,B 0,C 180,E1 -12670.85,E2 -12670.85} C_VEL
LIN {X 0,Y 372.43,Z 471.02,A -85,B 0,C 180,E1 -12671.572,E2 -12671.572} C_VEL
LIN {X 0,Y 373.535,Z 481.848,A -85,B 0,C 180,E1 -12672.376,E2 -12672.376} C_VEL
LIN {X 0,Y 372.41,Z 494.106,A -85,B 0,C 180,E1 -12673.418,E2 -12673.418} C_VEL
LIN {X 0,Y 371.302,Z 505.299,A -85,B 0,C 180,E1 -12674.636,E2 -12674.636} C_VEL
LIN {X 0,Y 370.377,Z 515.275,A -85,B 0,C 180,E1 -12676.002,E2 -12676.002} C_VEL
LIN {X 0,Y 369.542,Z 523.471,A -85,B 0,C 180,E1 -12677.369,E2 -12677.369} C_VEL
LIN {X 0,Y 368.69,Z 531.532,A -85,B 0,C 180,E1 -12679.013,E2 -12679.013} C_VEL
LIN {X 0,Y 368.165,Z 538.006,A -85,B 0,C 180,E1 -12680.664,E2 -12680.664} C_VEL
LIN {X 0,Y 367.793,Z 543.163,A -85,B 0,C 180,E1 -12682.315,E2 -12682.315} C_VEL
LIN {X 0,Y 367.601,Z 546.847,A -85,B 0,C 180,E1 -12683.809,E2 -12683.809} C_VEL
LIN {X 0,Y 367.519,Z 550.155,A -85,B 0,C 180,E1 -12685.615,E2 -12685.615} C_VEL
LIN {X 0,Y 367.51,Z 552.588,A -85,B 0,C 180,E1 -12687.81,E2 -12687.81} C_VEL
LIN {X 0,Y 367.546,Z 553.212,A -85,B 0,C 180,E1 -12688.906,E2 -12688.906} C_VEL
LIN {X 0,Y 367.538,Z 553.429,A -85,B 0,C 180,E1 -12690.002,E2 -12690.002} C_VEL
LIN {X 0,Y 367.547,Z 553.209,A -85,B 0,C 180,E1 -12691.098,E2 -12691.098} C_VEL
LIN {X 0,Y 367.525,Z 552.595,A -85,B 0,C 180,E1 -12692.194,E2 -12692.194} C_VEL
LIN {X 0,Y 367.447,Z 551.583,A -85,B 0,C 180,E1 -12693.291,E2 -12693.291} C_VEL
LIN {X 0,Y 367.519,Z 550.166,A -85,B 0,C 180,E1 -12694.389,E2 -12694.389} C_VEL
LIN {X 0,Y 367.6,Z 546.857,A -85,B 0,C 180,E1 -12696.189,E2 -12696.189} C_VEL
LIN {X 0,Y 367.895,Z 541.549,A -85,B 0,C 180,E1 -12698.239,E2 -12698.239} C_VEL
LIN {X 0,Y 368.346,Z 535.956,A -85,B 0,C 180,E1 -12699.89,E2 -12699.89} C_VEL
LIN {X 0,Y 368.931,Z 528.976,A -85,B 0,C 180,E1 -12701.54,E2 -12701.54} C_VEL
LIN {X 0,Y 369.896,Z 520.246,A -85,B 0,C 180,E1 -12703.181,E2 -12703.181} C_VEL
LIN {X 0,Y 370.844,Z 510.249,A -85,B 0,C 180,E1 -12704.694,E2 -12704.694} C_VEL
LIN {X 0,Y 371.746,Z 500.274,A -85,B 0,C 180,E1 -12705.912,E2 -12705.912} C_VEL
LIN {X 0,Y 372.821,Z 489.137,A -85,B 0,C 180,E1 -12706.991,E2 -12706.991} C_VEL
LIN {X 0,Y 373.494,Z 481.196,A -85,B 0,C 180,E1 -12707.623,E2 -12707.623} C_VEL
LIN {X 0,Y 372.147,Z 469.514,A -85,B 0,C 180,E1 -12708.458,E2 -12708.458} C_VEL
LIN {X 0,Y 370.264,Z 455.921,A -85,B 0,C 180,E1 -12709.199,E2 -12709.199} C_VEL
LIN {X 0,Y 368.444,Z 445.454,A -85,B 0,C 180,E1 -12709.646,E2 -12709.646} C_VEL
LIN {X 0,Y 368.907,Z 438.07,A -85,B 0,C 180,E1 -12712.99,E2 -12712.99} C_VEL
LIN {X 0,Y 369.516,Z 430.183,A -85,B 0,C 180,E1 -12716.63,E2 -12716.63} C_VEL
LIN {X 0,Y 370.225,Z 422.666,A -85,B 0,C 180,E1 -12720.204,E2 -12720.204} C_VEL
LIN {X 0,Y 370.916,Z 415.941,A -85,B 0,C 180,E1 -12723.519,E2 -12723.519} C_VEL
LIN {X 0,Y 371.46,Z 411.209,A -85,B 0,C 180,E1 -12725.912,E2 -12725.912} C_VEL
LIN {X 0,Y 371.206,Z 407.402,A -85,B 0,C 180,E1 -12727.976,E2 -12727.976} C_VEL
LIN {X 0,Y 370.118,Z 401.03,A -85,B 0,C 180,E1 -12731.653,E2 -12731.653} C_VEL
LIN {X 0,Y 369.074,Z 395.3,A -85,B 0,C 180,E1 -12735.205,E2 -12735.205} C_VEL
LIN {X 0,Y 368.915,Z 394.534,A -85,B 0,C 180,E1 -12735.833,E2 -12735.833} C_VEL
LIN {X 0,Y 368.918,Z 394.534,A -85,B 0,C 180,E1 -12739.644,E2 -12739.644} C_VEL
LIN {X 0,Y 368.907,Z 394.533,A -85,B 0,C 180,E1 -12743.145,E2 -12743.145} C_VEL
LIN {X 0,Y 368.903,Z 394.534,A -85,B 0,C 180,E1 -12746.462,E2 -12746.462} C_VEL
LIN {X 0,Y 368.936,Z 394.529,A -85,B 0,C 180,E1 -12749.047,E2 -12749.047} C_VEL
LIN {X 0,Y 368.97,Z 394.526,A -85,B 0,C 180,E1 -12752.797,E2 -12752.797} C_VEL
LIN {X 0,Y 368.952,Z 394.526,A -85,B 0,C 180,E1 -12756.113,E2 -12756.113} C_VEL
LIN {X 0,Y 368.943,Z 394.527,A -85,B 0,C 180,E1 -12759.947,E2 -12759.947} C_VEL
LIN {X 0,Y 368.982,Z 394.52,A -85,B 0,C 180,E1 -12763.399,E2 -12763.399} C_VEL
LIN {X 0,Y 369.064,Z 394.512,A -85,B 0,C 180,E1 -12766.79,E2 -12766.79} C_VEL
LIN {X 0,Y 369.074,Z 394.514,A -85,B 0,C 180,E1 -12770.132,E2 -12770.132} C_VEL
LIN {X 0,Y 369.205,Z 394.493,A -85,B 0,C 180,E1 -12773.442,E2 -12773.442} C_VEL
LIN {X 0,Y 369.321,Z 394.481,A -85,B 0,C 180,E1 -12777.819,E2 -12777.819} C_VEL
LIN {X 0,Y 369.462,Z 394.466,A -85,B 0,C 180,E1 -12780,E2 -12780} C_VEL
LIN {X 0,Y 369.322,Z 394.483,A -85,B 0,C 180,E1 -12782.181,E2 -12782.181} C_VEL
LIN {X 0,Y 369.206,Z 394.493,A -85,B 0,C 180,E1 -12786.648,E2 -12786.648} C_VEL
LIN {X 0,Y 369.144,Z 394.5,A -85,B 0,C 180,E1 -12788.761,E2 -12788.761} C_VEL
LIN {X 0,Y 369.011,Z 394.521,A -85,B 0,C 180,E1 -12792.093,E2 -12792.093} C_VEL
LIN {X 0,Y 369.004,Z 394.521,A -85,B 0,C 180,E1 -12795.465,E2 -12795.465} C_VEL
LIN {X 0,Y 368.964,Z 394.523,A -85,B 0,C 180,E1 -12798.894,E2 -12798.894} C_VEL
LIN {X 0,Y 368.938,Z 394.526,A -85,B 0,C 180,E1 -12802.395,E2 -12802.395} C_VEL
LIN {X 0,Y 369.006,Z 394.52,A -85,B 0,C 180,E1 -12805.98,E2 -12805.98} C_VEL
LIN {X 0,Y 368.921,Z 394.532,A -85,B 0,C 180,E1 -12809.69,E2 -12809.69} C_VEL
LIN {X 0,Y 368.903,Z 394.533,A -85,B 0,C 180,E1 -12813.042,E2 -12813.042} C_VEL
LIN {X 0,Y 368.923,Z 394.528,A -85,B 0,C 180,E1 -12816.196,E2 -12816.196} C_VEL
LIN {X 0,Y 368.909,Z 394.532,A -85,B 0,C 180,E1 -12818.952,E2 -12818.952} C_VEL
LIN {X 0,Y 368.887,Z 394.533,A -85,B 0,C 180,E1 -12822.009,E2 -12822.009} C_VEL
LIN {X 0,Y 368.931,Z 394.532,A -85,B 0,C 180,E1 -12825.182,E2 -12825.182} C_VEL
LIN {X 0,Y 368.888,Z 394.532,A -85,B 0,C 180,E1 -12828.177,E2 -12828.177} C_VEL
LIN {X 0,Y 368.915,Z 394.532,A -85,B 0,C 180,E1 -12831.359,E2 -12831.359} C_VEL
LIN {X 0,Y 368.942,Z 394.53,A -85,B 0,C 180,E1 -12835.145,E2 -12835.145} C_VEL
LIN {X 0,Y 368.935,Z 394.531,A -85,B 0,C 180,E1 -12839.045,E2 -12839.045} C_VEL
LIN {X 0,Y 368.968,Z 394.527,A -85,B 0,C 180,E1 -12842.795,E2 -12842.795} C_VEL
LIN {X 0,Y 368.95,Z 394.525,A -85,B 0,C 180,E1 -12846.111,E2 -12846.111} C_VEL
LIN {X 0,Y 368.941,Z 394.526,A -85,B 0,C 180,E1 -12849.946,E2 -12849.946} C_VEL
LIN {X 0,Y 368.98,Z 394.521,A -85,B 0,C 180,E1 -12853.397,E2 -12853.397} C_VEL
LIN {X 0,Y 369.024,Z 394.519,A -85,B 0,C 180,E1 -12856.787,E2 -12856.787} C_VEL
LIN {X 0,Y 368.739,Z 394.553,A -85,B 0,C 180,E1 -12860.121,E2 -12860.121} C_VEL
LIN {X 0,Y 368.535,Z 394.836,A -85,B 0,C 180,E1 -12862.327,E2 -12862.327} C_VEL
LIN {X 0,Y 368.54,Z 397.852,A -85,B 0,C 180,E1 -12865.623,E2 -12865.623} C_VEL
LIN {X 0,Y 368.049,Z 401.976,A -85,B 0,C 180,E1 -12869.998,E2 -12869.998} C_VEL
LIN {X 0,Y 368.2,Z 405.42,A -85,B 0,C 180,E1 -12873.554,E2 -12873.554} C_VEL
LIN {X 0,Y 372.143,Z 420.246,A -85,B 0,C 180,E1 -12874.364,E2 -12874.364} C_VEL
LIN {X 0,Y 374.583,Z 431.696,A -85,B 0,C 180,E1 -12875.158,E2 -12875.158} C_VEL
LIN {X 0,Y 373.789,Z 443.426,A -85,B 0,C 180,E1 -12876.028,E2 -12876.028} C_VEL
LIN {X 0,Y 372.917,Z 454.076,A -85,B 0,C 180,E1 -12877.034,E2 -12877.034} C_VEL
LIN {X 0,Y 371.907,Z 464.687,A -85,B 0,C 180,E1 -12878.282,E2 -12878.282} C_VEL
LIN {X 0,Y 370.982,Z 473.916,A -85,B 0,C 180,E1 -12879.633,E2 -12879.633} C_VEL
LIN {X 0,Y 370.048,Z 482.672,A -85,B 0,C 180,E1 -12881.223,E2 -12881.223} C_VEL
LIN {X 0,Y 369.287,Z 490.172,A -85,B 0,C 180,E1 -12882.919,E2 -12882.919} C_VEL
LIN {X 0,Y 368.738,Z 495.242,A -85,B 0,C 180,E1 -12884.343,E2 -12884.343} C_VEL
LIN {X 0,Y 368.273,Z 500.14,A -85,B 0,C 180,E1 -12886.062,E2 -12886.062} C_VEL
LIN {X 0,Y 367.902,Z 503.87,A -85,B 0,C 180,E1 -12887.794,E2 -12887.794} C_VEL
LIN {X 0,Y 367.695,Z 505.734,A -85,B 0,C 180,E1 -12888.959,E2 -12888.959} C_VEL
LIN {X 0,Y 367.53,Z 507.464,A -85,B 0,C 180,E1 -12890.448,E2 -12890.448} C_VEL
LIN {X 0,Y 367.445,Z 508.587,A -85,B 0,C 180,E1 -12892.488,E2 -12892.488} C_VEL
LIN {X 0,Y 367.441,Z 508.623,A -85,B 0,C 180,E1 -12893.679,E2 -12893.679} C_VEL
LIN {X 0,Y 367.493,Z 508.216,A -85,B 0,C 180,E1 -12894.878,E2 -12894.878} C_VEL
LIN {X 0,Y 367.628,Z 507.282,A -85,B 0,C 180,E1 -12896.081,E2 -12896.081} C_VEL
LIN {X 0,Y 367.807,Z 505.884,A -85,B 0,C 180,E1 -12897.293,E2 -12897.293} C_VEL
LIN {X 0,Y 368.155,Z 502.795,A -85,B 0,C 180,E1 -12899.126,E2 -12899.126} C_VEL
LIN {X 0,Y 368.596,Z 498.356,A -85,B 0,C 180,E1 -12900.981,E2 -12900.981} C_VEL
LIN {X 0,Y 369.231,Z 492.676,A -85,B 0,C 180,E1 -12902.769,E2 -12902.769} C_VEL
LIN {X 0,Y 370.013,Z 486.094,A -85,B 0,C 180,E1 -12904.404,E2 -12904.404} C_VEL
LIN {X 0,Y 370.882,Z 478.275,A -85,B 0,C 180,E1 -12905.972,E2 -12905.972} C_VEL
LIN {X 0,Y 371.275,Z 474.653,A -85,B 0,C 180,E1 -12906.594,E2 -12906.594} C_VEL
LIN {X 0,Y 371.089,Z 470.668,A -85,B 0,C 180,E1 -12907.269,E2 -12907.269} C_VEL
LIN {X 0,Y 369.023,Z 463.968,A -85,B 0,C 180,E1 -12908.361,E2 -12908.361} C_VEL
LIN {X 0,Y 366.985,Z 456.73,A -85,B 0,C 180,E1 -12909.366,E2 -12909.366} C_VEL
LIN {X 0,Y 366.83,Z 451.908,A -85,B 0,C 180,E1 -12909.896,E2 -12909.896} C_VEL
LIN {X 0,Y 367.866,Z 439.939,A -85,B 0,C 180,E1 -12910.956,E2 -12910.956} C_VEL
LIN {X 0,Y 368.223,Z 433.963,A -85,B 0,C 180,E1 -12911.395,E2 -12911.395} C_VEL
LIN {X 0,Y 365.475,Z 422.055,A -85,B 0,C 180,E1 -12912.298,E2 -12912.298} C_VEL
LIN {X 0,Y 361.803,Z 409.517,A -85,B 0,C 180,E1 -12913.065,E2 -12913.065} C_VEL
LIN {X 0,Y 361.056,Z 406.875,A -85,B 0,C 180,E1 -12913.227,E2 -12913.227} C_VEL
LIN {X 0,Y 361.156,Z 403.43,A -85,B 0,C 180,E1 -12917.071,E2 -12917.071} C_VEL
LIN {X 0,Y 361.234,Z 400.805,A -85,B 0,C 180,E1 -12920.056,E2 -12920.056} C_VEL
LIN {X 0,Y 361.368,Z 398.328,A -85,B 0,C 180,E1 -12922.922,E2 -12922.922} C_VEL
LIN {X 0,Y 361.483,Z 396.002,A -85,B 0,C 180,E1 -12925.68,E2 -12925.68} C_VEL
LIN {X 0,Y 361.61,Z 395.449,A -85,B 0,C 180,E1 -12927.031,E2 -12927.031} C_VEL
LIN {X 0,Y 361.819,Z 395.42,A -85,B 0,C 180,E1 -12929.667,E2 -12929.667} C_VEL
LIN {X 0,Y 361.924,Z 395.404,A -85,B 0,C 180,E1 -12933.277,E2 -12933.277} C_VEL
LIN {X 0,Y 361.905,Z 395.407,A -85,B 0,C 180,E1 -12937.146,E2 -12937.146} C_VEL
LIN {X 0,Y 361.916,Z 395.405,A -85,B 0,C 180,E1 -12940.724,E2 -12940.724} C_VEL
LIN {X 0,Y 361.927,Z 395.401,A -85,B 0,C 180,E1 -12944.225,E2 -12944.225} C_VEL
LIN {X 0,Y 361.981,Z 395.394,A -85,B 0,C 180,E1 -12946.527,E2 -12946.527} C_VEL
LIN {X 0,Y 362.017,Z 395.389,A -85,B 0,C 180,E1 -12949.938,E2 -12949.938} C_VEL
LIN {X 0,Y 362.132,Z 395.377,A -85,B 0,C 180,E1 -12952.192,E2 -12952.192} C_VEL
LIN {X 0,Y 362.105,Z 395.381,A -85,B 0,C 180,E1 -12954.431,E2 -12954.431} C_VEL
LIN {X 0,Y 362.264,Z 395.361,A -85,B 0,C 180,E1 -12957.776,E2 -12957.776} C_VEL
LIN {X 0,Y 362.409,Z 395.342,A -85,B 0,C 180,E1 -12960,E2 -12960} C_VEL
LIN {X 0,Y 362.27,Z 395.36,A -85,B 0,C 180,E1 -12962.224,E2 -12962.224} C_VEL
LIN {X 0,Y 362.152,Z 395.375,A -85,B 0,C 180,E1 -12966.687,E2 -12966.687} C_VEL
LIN {X 0,Y 362.056,Z 395.387,A -85,B 0,C 180,E1 -12968.934,E2 -12968.934} C_VEL
LIN {X 0,Y 361.947,Z 395.4,A -85,B 0,C 180,E1 -12972.333,E2 -12972.333} C_VEL
LIN {X 0,Y 361.943,Z 395.402,A -85,B 0,C 180,E1 -12974.621,E2 -12974.621} C_VEL
LIN {X 0,Y 361.943,Z 395.402,A -85,B 0,C 180,E1 -12978.1,E2 -12978.1} C_VEL
LIN {X 0,Y 361.914,Z 395.406,A -85,B 0,C 180,E1 -12981.652,E2 -12981.652} C_VEL
LIN {X 0,Y 361.913,Z 395.409,A -85,B 0,C 180,E1 -12985.291,E2 -12985.291} C_VEL
LIN {X 0,Y 361.891,Z 395.411,A -85,B 0,C 180,E1 -12987.781,E2 -12987.781} C_VEL
LIN {X 0,Y 361.822,Z 395.419,A -85,B 0,C 180,E1 -12991.631,E2 -12991.631} C_VEL
LIN {X 0,Y 361.86,Z 395.412,A -85,B 0,C 180,E1 -12995.347,E2 -12995.347} C_VEL
LIN {X 0,Y 361.861,Z 395.414,A -85,B 0,C 180,E1 -12999.03,E2 -12999.03} C_VEL
LIN {X 0,Y 361.874,Z 395.417,A -85,B 0,C 180,E1 -13002.443,E2 -13002.443} C_VEL
LIN {X 0,Y 361.926,Z 395.51,A -85,B 0,C 180,E1 -13003.312,E2 -13003.312} C_VEL
LIN {X 0,Y 362.744,Z 400.119,A -85,B 0,C 180,E1 -13006.577,E2 -13006.577} C_VEL
LIN {X 0,Y 363.615,Z 404.903,A -85,B 0,C 180,E1 -13009.686,E2 -13009.686} C_VEL
LIN {X 0,Y 364.317,Z 409.179,A -85,B 0,C 180,E1 -13012.272,E2 -13012.272} C_VEL
LIN {X 0,Y 364.439,Z 412.378,A -85,B 0,C 180,E1 -13014.091,E2 -13014.091} C_VEL
LIN {X 0,Y 363.823,Z 417.299,A -85,B 0,C 180,E1 -13016.688,E2 -13016.688} C_VEL
LIN {X 0,Y 362.965,Z 425.015,A -85,B 0,C 180,E1 -13020.613,E2 -13020.613} C_VEL
LIN {X 0,Y 362.305,Z 432.227,A -85,B 0,C 180,E1 -13024.125,E2 -13024.125} C_VEL
LIN {X 0,Y 361.594,Z 441.202,A -85,B 0,C 180,E1 -13028.331,E2 -13028.331} C_VEL
LIN {X 0,Y 361.418,Z 444.534,A -85,B 0,C 180,E1 -13029.825,E2 -13029.825} C_VEL
LIN {X 0,Y 363.908,Z 458.098,A -85,B 0,C 180,E1 -13030.443,E2 -13030.443} C_VEL
LIN {X 0,Y 365.551,Z 471.356,A -85,B 0,C 180,E1 -13031.251,E2 -13031.251} C_VEL
LIN {X 0,Y 366.671,Z 482.886,A -85,B 0,C 180,E1 -13032.144,E2 -13032.144} C_VEL
LIN {X 0,Y 365.599,Z 493.782,A -85,B 0,C 180,E1 -13033.1,E2 -13033.1} C_VEL
LIN {X 0,Y 364.443,Z 504.944,A -85,B 0,C 180,E1 -13034.339,E2 -13034.339} C_VEL
LIN {X 0,Y 363.471,Z 514.906,A -85,B 0,C 180,E1 -13035.73,E2 -13035.73} C_VEL
LIN {X 0,Y 362.406,Z 524.583,A -85,B 0,C 180,E1 -13037.401,E2 -13037.401} C_VEL
LIN {X 0,Y 361.586,Z 532.298,A -85,B 0,C 180,E1 -13039.078,E2 -13039.078} C_VEL
LIN {X 0,Y 360.969,Z 539.446,A -85,B 0,C 180,E1 -13041.042,E2 -13041.042} C_VEL
LIN {X 0,Y 360.678,Z 544.209,A -85,B 0,C 180,E1 -13042.726,E2 -13042.726} C_VEL
LIN {X 0,Y 360.477,Z 547.853,A -85,B 0,C 180,E1 -13044.408,E2 -13044.408} C_VEL
LIN {X 0,Y 360.45,Z 549.734,A -85,B 0,C 180,E1 -13045.529,E2 -13045.529} C_VEL
LIN {X 0,Y 360.414,Z 552.161,A -85,B 0,C 180,E1 -13047.767,E2 -13047.767} C_VEL
LIN {X 0,Y 360.482,Z 552.785,A -85,B 0,C 180,E1 -13048.885,E2 -13048.885} C_VEL
LIN {X 0,Y 360.474,Z 552.999,A -85,B 0,C 180,E1 -13050.002,E2 -13050.002} C_VEL
LIN {X 0,Y 360.483,Z 552.777,A -85,B 0,C 180,E1 -13051.119,E2 -13051.119} C_VEL
LIN {X 0,Y 360.429,Z 552.159,A -85,B 0,C 180,E1 -13052.237,E2 -13052.237} C_VEL
LIN {X 0,Y 360.364,Z 551.145,A -85,B 0,C 180,E1 -13053.356,E2 -13053.356} C_VEL
LIN {X 0,Y 360.451,Z 549.723,A -85,B 0,C 180,E1 -13054.475,E2 -13054.475} C_VEL
LIN {X 0,Y 360.529,Z 546.683,A -85,B 0,C 180,E1 -13056.186,E2 -13056.186} C_VEL
LIN {X 0,Y 360.721,Z 542.708,A -85,B 0,C 180,E1 -13057.841,E2 -13057.841} C_VEL
LIN {X 0,Y 361.227,Z 536.504,A -85,B 0,C 180,E1 -13059.804,E2 -13059.804} C_VEL
LIN {X 0,Y 361.826,Z 529.739,A -85,B 0,C 180,E1 -13061.486,E2 -13061.486} C_VEL
LIN {X 0,Y 362.793,Z 521.364,A -85,B 0,C 180,E1 -13063.159,E2 -13063.159} C_VEL
LIN {X 0,Y 363.774,Z 511.633,A -85,B 0,C 180,E1 -13064.709,E2 -13064.709} C_VEL
LIN {X 0,Y 364.756,Z 500.935,A -85,B 0,C 180,E1 -13066.081,E2 -13066.081} C_VEL
LIN {X 0,Y 365.865,Z 490.143,A -85,B 0,C 180,E1 -13067.18,E2 -13067.18} C_VEL
LIN {X 0,Y 366.566,Z 481.839,A -85,B 0,C 180,E1 -13067.866,E2 -13067.866} C_VEL
LIN {X 0,Y 365.205,Z 469.596,A -85,B 0,C 180,E1 -13068.778,E2 -13068.778} C_VEL
LIN {X 0,Y 363.364,Z 456.172,A -85,B 0,C 180,E1 -13069.537,E2 -13069.537} C_VEL
LIN {X 0,Y 361.43,Z 445.069,A -85,B 0,C 180,E1 -13070.024,E2 -13070.024} C_VEL
LIN {X 0,Y 361.893,Z 437.655,A -85,B 0,C 180,E1 -13073.462,E2 -13073.462} C_VEL
LIN {X 0,Y 362.489,Z 430.409,A -85,B 0,C 180,E1 -13076.892,E2 -13076.892} C_VEL
LIN {X 0,Y 363.181,Z 423.579,A -85,B 0,C 180,E1 -13080.209,E2 -13080.209} C_VEL
LIN {X 0,Y 363.842,Z 417.391,A -85,B 0,C 180,E1 -13083.313,E2 -13083.313} C_VEL
LIN {X 0,Y 364.439,Z 412.381,A -85,B 0,C 180,E1 -13085.909,E2 -13085.909} C_VEL
LIN {X 0,Y 364.185,Z 408.327,A -85,B 0,C 180,E1 -13088.138,E2 -13088.138} C_VEL
LIN {X 0,Y 363.108,Z 402.043,A -85,B 0,C 180,E1 -13091.861,E2 -13091.861} C_VEL
LIN {X 0,Y 362.017,Z 396.063,A -85,B 0,C 180,E1 -13095.662,E2 -13095.662} C_VEL
LIN {X 0,Y 361.873,Z 395.411,A -85,B 0,C 180,E1 -13096.24,E2 -13096.24} C_VEL
LIN {X 0,Y 361.861,Z 395.411,A -85,B 0,C 180,E1 -13100.139,E2 -13100.139} C_VEL
LIN {X 0,Y 361.873,Z 395.41,A -85,B 0,C 180,E1 -13102.982,E2 -13102.982} C_VEL
LIN {X 0,Y 361.865,Z 395.412,A -85,B 0,C 180,E1 -13106.631,E2 -13106.631} C_VEL
LIN {X 0,Y 361.88,Z 395.405,A -85,B 0,C 180,E1 -13109.672,E2 -13109.672} C_VEL
LIN {X 0,Y 361.961,Z 395.395,A -85,B 0,C 180,E1 -13113.475,E2 -13113.475} C_VEL
LIN {X 0,Y 361.897,Z 395.404,A -85,B 0,C 180,E1 -13117.145,E2 -13117.145} C_VEL
LIN {X 0,Y 361.913,Z 395.404,A -85,B 0,C 180,E1 -13120.724,E2 -13120.724} C_VEL
LIN {X 0,Y 361.939,Z 395.398,A -85,B 0,C 180,E1 -13123.066,E2 -13123.066} C_VEL
LIN {X 0,Y 362.006,Z 395.394,A -85,B 0,C 180,E1 -13126.528,E2 -13126.528} C_VEL
LIN {X 0,Y 362.038,Z 395.388,A -85,B 0,C 180,E1 -13129.938,E2 -13129.938} C_VEL
LIN {X 0,Y 362.167,Z 395.369,A -85,B 0,C 180,E1 -13133.314,E2 -13133.314} C_VEL
LIN {X 0,Y 362.285,Z 395.357,A -85,B 0,C 180,E1 -13137.776,E2 -13137.776} C_VEL
LIN {X 0,Y 362.432,Z 395.341,A -85,B 0,C 180,E1 -13140,E2 -13140} C_VEL
LIN {X 0,Y 362.286,Z 395.359,A -85,B 0,C 180,E1 -13142.223,E2 -13142.223} C_VEL
LIN {X 0,Y 362.176,Z 395.368,A -85,B 0,C 180,E1 -13146.686,E2 -13146.686} C_VEL
LIN {X 0,Y 362.08,Z 395.38,A -85,B 0,C 180,E1 -13148.933,E2 -13148.933} C_VEL
LIN {X 0,Y 361.966,Z 395.396,A -85,B 0,C 180,E1 -13152.332,E2 -13152.332} C_VEL
LIN {X 0,Y 361.968,Z 395.394,A -85,B 0,C 180,E1 -13154.62,E2 -13154.62} C_VEL
LIN {X 0,Y 361.962,Z 395.397,A -85,B 0,C 180,E1 -13158.099,E2 -13158.099} C_VEL
LIN {X 0,Y 361.898,Z 395.408,A -85,B 0,C 180,E1 -13161.652,E2 -13161.652} C_VEL
LIN {X 0,Y 361.935,Z 395.401,A -85,B 0,C 180,E1 -13165.29,E2 -13165.29} C_VEL
LIN {X 0,Y 361.914,Z 395.404,A -85,B 0,C 180,E1 -13167.778,E2 -13167.778} C_VEL
LIN {X 0,Y 361.844,Z 395.414,A -85,B 0,C 180,E1 -13171.629,E2 -13171.629} C_VEL
LIN {X 0,Y 361.88,Z 395.41,A -85,B 0,C 180,E1 -13175.344,E2 -13175.344} C_VEL
LIN {X 0,Y 361.875,Z 395.409,A -85,B 0,C 180,E1 -13179.026,E2 -13179.026} C_VEL
LIN {X 0,Y 361.842,Z 395.412,A -85,B 0,C 180,E1 -13182.828,E2 -13182.828} C_VEL
LIN {X 0,Y 361.84,Z 395.41,A -85,B 0,C 180,E1 -13185.943,E2 -13185.943} C_VEL
LIN {X 0,Y 361.841,Z 395.415,A -85,B 0,C 180,E1 -13189.244,E2 -13189.244} C_VEL
LIN {X 0,Y 361.869,Z 395.41,A -85,B 0,C 180,E1 -13192.776,E2 -13192.776} C_VEL
LIN {X 0,Y 361.86,Z 395.408,A -85,B 0,C 180,E1 -13195.718,E2 -13195.718} C_VEL
LIN {X 0,Y 361.878,Z 395.405,A -85,B 0,C 180,E1 -13199.671,E2 -13199.671} C_VEL
LIN {X 0,Y 361.959,Z 395.396,A -85,B 0,C 180,E1 -13203.474,E2 -13203.474} C_VEL
LIN {X 0,Y 361.895,Z 395.406,A -85,B 0,C 180,E1 -13207.143,E2 -13207.143} C_VEL
LIN {X 0,Y 361.911,Z 395.407,A -85,B 0,C 180,E1 -13210.722,E2 -13210.722} C_VEL
LIN {X 0,Y 361.937,Z 395.4,A -85,B 0,C 180,E1 -13213.064,E2 -13213.064} C_VEL
LIN {X 0,Y 361.975,Z 395.398,A -85,B 0,C 180,E1 -13216.525,E2 -13216.525} C_VEL
LIN {X 0,Y 361.697,Z 395.429,A -85,B 0,C 180,E1 -13219.927,E2 -13219.927} C_VEL
LIN {X 0,Y 361.502,Z 395.578,A -85,B 0,C 180,E1 -13222.176,E2 -13222.176} C_VEL
LIN {X 0,Y 361.506,Z 398.614,A -85,B 0,C 180,E1 -13225.538,E2 -13225.538} C_VEL
LIN {X 0,Y 360.994,Z 402.804,A -85,B 0,C 180,E1 -13229.998,E2 -13229.998} C_VEL
LIN {X 0,Y 361.141,Z 405.768,A -85,B 0,C 180,E1 -13233.17,E2 -13233.17} C_VEL
LIN {X 0,Y 365.075,Z 420.535,A -85,B 0,C 180,E1 -13233.999,E2 -13233.999} C_VEL
LIN {X 0,Y 367.362,Z 430.801,A -85,B 0,C 180,E1 -13234.725,E2 -13234.725} C_VEL
LIN {X 0,Y 367.709,Z 433.922,A -85,B 0,C 180,E1 -13234.96,E2 -13234.96} C_VEL
LIN {X 0,Y 366.864,Z 445.964,A -85,B 0,C 180,E1 -13235.907,E2 -13235.907} C_VEL
LIN {X 0,Y 366.018,Z 455.834,A -85,B 0,C 180,E1 -13236.89,E2 -13236.89} C_VEL
LIN {X 0,Y 364.925,Z 466.195,A -85,B 0,C 180,E1 -13238.163,E2 -13238.163} C_VEL
LIN {X 0,Y 363.874,Z 475.9,A -85,B 0,C 180,E1 -13239.657,E2 -13239.657} C_VEL
LIN {X 0,Y 363.004,Z 483.831,A -85,B 0,C 180,E1 -13241.161,E2 -13241.161} C_VEL
LIN {X 0,Y 362.233,Z 491.188,A -85,B 0,C 180,E1 -13242.89,E2 -13242.89} C_VEL
LIN {X 0,Y 361.585,Z 497.033,A -85,B 0,C 180,E1 -13244.633,E2 -13244.633} C_VEL
LIN {X 0,Y 361.144,Z 501.606,A -85,B 0,C 180,E1 -13246.388,E2 -13246.388} C_VEL
LIN {X 0,Y 360.76,Z 505.051,A -85,B 0,C 180,E1 -13248.159,E2 -13248.159} C_VEL
LIN {X 0,Y 360.555,Z 506.761,A -85,B 0,C 180,E1 -13249.349,E2 -13249.349} C_VEL
LIN {X 0,Y 360.426,Z 508.055,A -85,B 0,C 180,E1 -13250.616,E2 -13250.616} C_VEL
LIN {X 0,Y 360.376,Z 508.761,A -85,B 0,C 180,E1 -13251.746,E2 -13251.746} C_VEL
LIN {X 0,Y 360.373,Z 509.072,A -85,B 0,C 180,E1 -13253.567,E2 -13253.567} C_VEL
LIN {X 0,Y 360.465,Z 508.334,A -85,B 0,C 180,E1 -13255.397,E2 -13255.397} C_VEL
LIN {X 0,Y 360.633,Z 507.26,A -85,B 0,C 180,E1 -13256.627,E2 -13256.627} C_VEL
LIN {X 0,Y 361.024,Z 504.021,A -85,B 0,C 180,E1 -13258.835,E2 -13258.835} C_VEL
LIN {X 0,Y 361.479,Z 499.725,A -85,B 0,C 180,E1 -13260.796,E2 -13260.796} C_VEL
LIN {X 0,Y 362.113,Z 494.472,A -85,B 0,C 180,E1 -13262.584,E2 -13262.584} C_VEL
LIN {X 0,Y 362.855,Z 488.561,A -85,B 0,C 180,E1 -13264.169,E2 -13264.169} C_VEL
LIN {X 0,Y 363.746,Z 480.608,A -85,B 0,C 180,E1 -13265.877,E2 -13265.877} C_VEL
LIN {X 0,Y 364.764,Z 472.007,A -85,B 0,C 180,E1 -13267.363,E2 -13267.363} C_VEL
LIN {X 0,Y 365.722,Z 462.938,A -85,B 0,C 180,E1 -13268.645,E2 -13268.645} C_VEL
LIN {X 0,Y 366.83,Z 451.908,A -85,B 0,C 180,E1 -13269.896,E2 -13269.896} C_VEL
LIN {X 0,Y 366.712,Z 446.952,A -85,B 0,C 180,E1 -13270.402,E2 -13270.402} C_VEL
LIN {X 0,Y 365.532,Z 442.072,A -85,B 0,C 180,E1 -13270.915,E2 -13270.915} C_VEL
LIN {X 0,Y 361.68,Z 432.438,A -85,B 0,C 180,E1 -13271.898,E2 -13271.898} C_VEL
LIN {X 0,Y 359.337,Z 425.606,A -85,B 0,C 180,E1 -13272.478,E2 -13272.478} C_VEL
LIN {X 0,Y 355.736,Z 412.929,A -85,B 0,C 180,E1 -13273.332,E2 -13273.332} C_VEL
LIN {X 0,Y 354.032,Z 407.335,A -85,B 0,C 180,E1 -13273.661,E2 -13273.661} C_VEL
LIN {X 0,Y 354.128,Z 404.177,A -85,B 0,C 180,E1 -13277.243,E2 -13277.243} C_VEL
LIN {X 0,Y 354.232,Z 401.203,A -85,B 0,C 180,E1 -13280.688,E2 -13280.688} C_VEL
LIN {X 0,Y 354.405,Z 398.071,A -85,B 0,C 180,E1 -13284.389,E2 -13284.389} C_VEL
LIN {X 0,Y 354.471,Z 396.447,A -85,B 0,C 180,E1 -13286.374,E2 -13286.374} C_VEL
LIN {X 0,Y 354.733,Z 396.303,A -85,B 0,C 180,E1 -13288.995,E2 -13288.995} C_VEL
LIN {X 0,Y 354.829,Z 396.288,A -85,B 0,C 180,E1 -13291.617,E2 -13291.617} C_VEL
LIN {X 0,Y 354.883,Z 396.282,A -85,B 0,C 180,E1 -13294.171,E2 -13294.171} C_VEL
LIN {X 0,Y 354.874,Z 396.282,A -85,B 0,C 180,E1 -13297.897,E2 -13297.897} C_VEL
LIN {X 0,Y 354.905,Z 396.276,A -85,B 0,C 180,E1 -13301.89,E2 -13301.89} C_VEL
LIN {X 0,Y 354.924,Z 396.276,A -85,B 0,C 180,E1 -13305.98,E2 -13305.98} C_VEL
LIN {X 0,Y 354.963,Z 396.268,A -85,B 0,C 180,E1 -13309.736,E2 -13309.736} C_VEL
LIN {X 0,Y 355.095,Z 396.253,A -85,B 0,C 180,E1 -13312.037,E2 -13312.037} C_VEL
LIN {X 0,Y 355.079,Z 396.257,A -85,B 0,C 180,E1 -13314.321,E2 -13314.321} C_VEL
LIN {X 0,Y 355.227,Z 396.237,A -85,B 0,C 180,E1 -13317.732,E2 -13317.732} C_VEL
LIN {X 0,Y 355.379,Z 396.218,A -85,B 0,C 180,E1 -13320,E2 -13320} C_VEL
LIN {X 0,Y 355.234,Z 396.237,A -85,B 0,C 180,E1 -13322.268,E2 -13322.268} C_VEL
LIN {X 0,Y 355.118,Z 396.251,A -85,B 0,C 180,E1 -13326.82,E2 -13326.82} C_VEL
LIN {X 0,Y 354.997,Z 396.266,A -85,B 0,C 180,E1 -13329.113,E2 -13329.113} C_VEL
LIN {X 0,Y 354.907,Z 396.277,A -85,B 0,C 180,E1 -13332.582,E2 -13332.582} C_VEL
LIN {X 0,Y 354.871,Z 396.282,A -85,B 0,C 180,E1 -13336.097,E2 -13336.097} C_VEL
LIN {X 0,Y 354.892,Z 396.281,A -85,B 0,C 180,E1 -13338.473,E2 -13338.473} C_VEL
LIN {X 0,Y 354.874,Z 396.283,A -85,B 0,C 180,E1 -13342.104,E2 -13342.104} C_VEL
LIN {X 0,Y 354.883,Z 396.283,A -85,B 0,C 180,E1 -13345.829,E2 -13345.829} C_VEL
LIN {X 0,Y 354.801,Z 396.294,A -85,B 0,C 180,E1 -13349.684,E2 -13349.684} C_VEL
LIN {X 0,Y 354.791,Z 396.293,A -85,B 0,C 180,E1 -13353.704,E2 -13353.704} C_VEL
LIN {X 0,Y 354.785,Z 396.293,A -85,B 0,C 180,E1 -13356.461,E2 -13356.461} C_VEL
LIN {X 0,Y 354.81,Z 396.292,A -85,B 0,C 180,E1 -13359.426,E2 -13359.426} C_VEL
LIN {X 0,Y 354.856,Z 396.371,A -85,B 0,C 180,E1 -13362.785,E2 -13362.785} C_VEL
LIN {X 0,Y 355.501,Z 399.871,A -85,B 0,C 180,E1 -13365.373,E2 -13365.373} C_VEL
LIN {X 0,Y 356.57,Z 405.878,A -85,B 0,C 180,E1 -13369.43,E2 -13369.43} C_VEL
LIN {X 0,Y 357.347,Z 410.732,A -85,B 0,C 180,E1 -13372.437,E2 -13372.437} C_VEL
LIN {X 0,Y 357.324,Z 414.395,A -85,B 0,C 180,E1 -13374.538,E2 -13374.538} C_VEL
LIN {X 0,Y 356.505,Z 420.826,A -85,B 0,C 180,E1 -13377.961,E2 -13377.961} C_VEL
LIN {X 0,Y 355.824,Z 426.836,A -85,B 0,C 180,E1 -13381.062,E2 -13381.062} C_VEL
LIN {X 0,Y 355.088,Z 434.436,A -85,B 0,C 180,E1 -13384.819,E2 -13384.819} C_VEL
LIN {X 0,Y 354.405,Z 443.352,A -85,B 0,C 180,E1 -13389.09,E2 -13389.09} C_VEL
LIN {X 0,Y 354.374,Z 443.913,A -85,B 0,C 180,E1 -13389.354,E2 -13389.354} C_VEL
LIN {X 0,Y 357.107,Z 458.685,A -85,B 0,C 180,E1 -13390.084,E2 -13390.084} C_VEL
LIN {X 0,Y 358.782,Z 472.547,A -85,B 0,C 180,E1 -13390.972,E2 -13390.972} C_VEL
LIN {X 0,Y 359.771,Z 484.388,A -85,B 0,C 180,E1 -13391.937,E2 -13391.937} C_VEL
LIN {X 0,Y 358.485,Z 496.156,A -85,B 0,C 180,E1 -13393.048,E2 -13393.048} C_VEL
LIN {X 0,Y 357.362,Z 506.331,A -85,B 0,C 180,E1 -13394.258,E2 -13394.258} C_VEL
LIN {X 0,Y 356.343,Z 516.331,A -85,B 0,C 180,E1 -13395.73,E2 -13395.73} C_VEL
LIN {X 0,Y 355.276,Z 525.574,A -85,B 0,C 180,E1 -13397.434,E2 -13397.434} C_VEL
LIN {X 0,Y 354.477,Z 533.037,A -85,B 0,C 180,E1 -13399.146,E2 -13399.146} C_VEL
LIN {X 0,Y 353.921,Z 539.044,A -85,B 0,C 180,E1 -13400.862,E2 -13400.862} C_VEL
LIN {X 0,Y 353.61,Z 543.801,A -85,B 0,C 180,E1 -13402.58,E2 -13402.58} C_VEL
